  MoveL 1332 to (515.77, 1197.49, 513.19) mm, rotated rx -180 ry 0 rz -88.32 deg; joints [33.086, -49.843, -64.366, 36.804, -42.297, -55.101]
  MoveL 1333 to (513.37, 1199.03, 513.19) mm, rotated rx -180 ry 0 rz -88.32 deg; joints [32.917, -49.844, -64.366, 36.702, -42.2, -54.906]
  MoveL 1334 to (510.99, 1200.59, 513.19) mm, rotated rx -180 ry 0 rz -88.32 deg; joints [32.749, -49.843, -64.366, 36.6, -42.102, -54.711]
  MoveL 1335 to (508.6, 1202.15, 513.19) mm, rotated rx 180 ry 0 rz -88.32 deg; joints [32.58, -49.841, -64.365, 36.498, -42.004, -54.517]
  MoveL 1336 to (506.22, 1203.72, 513.19) mm, rotated rx -180 ry 0 rz -88.32 deg; joints [32.411, -49.837, -64.363, 36.396, -41.905, -54.322]
  MoveL 1337 to (503.85, 1205.29, 513.19) mm, rotated rx 180 ry 0 rz -88.32 deg; joints [32.243, -49.831, -64.361, 36.293, -41.806, -54.128]
  MoveL 1338 to (501.47, 1206.87, 513.19) mm, rotated rx -180 ry 0 rz -88.32 deg; joints [32.074, -49.825, -64.357, 36.19, -41.707, -53.934]
  MoveL 1339 to (499.11, 1208.46, 513.19) mm, rotated rx -180 ry 0 rz -88.32 deg; joints [31.906, -49.816, -64.354, 36.088, -41.607, -53.739]
  MoveL 1340 to (496.75, 1210.05, 513.19) mm, rotated rx -180 ry 0 rz -88.32 deg; joints [31.737, -49.807, -64.349, 35.985, -41.507, -53.545]
  MoveL 1341 to (494.39, 1211.65, 513.19) mm, rotated rx -180 ry 0 rz -88.32 deg; joints [31.569, -49.796, -64.344, 35.881, -41.406, -53.351]
  MoveL 1342 to (492.03, 1213.26, 513.19) mm, rotated rx -180 ry 0 rz -88.32 deg; joints [31.401, -49.783, -64.338, 35.778, -41.305, -53.157]
  MoveL 1343 to (489.69, 1214.88, 513.19) mm, rotated rx -180 ry 0 rz -88.32 deg; joints [31.233, -49.769, -64.332, 35.675, -41.204, -52.963]
  MoveL 1344 to (487.34, 1216.5, 513.19) mm, rotated rx -180 ry 0 rz -88.32 deg; joints [31.064, -49.754, -64.324, 35.571, -41.103, -52.77]
  MoveL 1345 to (485, 1218.12, 513.19) mm, rotated rx -180 ry 0 rz -88.32 deg; joints [30.896, -49.737, -64.316, 35.468, -41.001, -52.576]
  MoveL 1346 to (482.67, 1219.76, 513.19) mm, rotated rx -180 ry 0 rz -88.32 deg; joints [30.728, -49.718, -64.308, 35.364, -40.899, -52.383]
  MoveL 1347 to (480.34, 1221.4, 513.19) mm, rotated rx 180 ry 0 rz -88.32 deg; joints [30.561, -49.698, -64.299, 35.26, -40.796, -52.189]
  MoveL 1348 to (478.01, 1223.04, 513.19) mm, rotated rx -180 ry 0 rz -88.32 deg; joints [30.393, -49.677, -64.289, 35.156, -40.693, -51.996]
  MoveL 1349 to (475.69, 1224.7, 513.19) mm, rotated rx -180 ry 0 rz -88.32 deg; joints [30.225, -49.655, -64.278, 35.052, -40.59, -51.803]
  MoveL 1350 to (473.37, 1226.36, 513.19) mm, rotated rx -180 ry 0 rz -88.32 deg; joints [30.058, -49.631, -64.267, 34.947, -40.487, -51.61]
  MoveL 1351 to (471.06, 1228.02, 513.19) mm, rotated rx 180 ry 0 rz -88.32 deg; joints [29.891, -49.605, -64.255, 34.843, -40.383, -51.418]
  MoveL 1352 to (468.75, 1229.7, 513.19) mm, rotated rx -180 ry 0 rz -88.32 deg; joints [29.723, -49.578, -64.243, 34.739, -40.279, -51.225]
  MoveL 1353 to (466.45, 1231.38, 513.19) mm, rotated rx -180 ry 0 rz -88.32 deg; joints [29.556, -49.55, -64.229, 34.634, -40.175, -51.033]
  MoveL 1354 to (464.15, 1233.06, 513.19) mm, rotated rx -180 ry 0 rz -88.32 deg; joints [29.39, -49.52, -64.216, 34.529, -40.07, -50.841]
  MoveL 1355 to (461.86, 1234.75, 513.19) mm, rotated rx -180 ry 0 rz -88.32 deg; joints [29.223, -49.489, -64.201, 34.425, -39.965, -50.649]
  MoveL 1356 to (459.57, 1236.45, 513.19) mm, rotated rx -180 ry 0 rz -88.32 deg; joints [29.056, -49.456, -64.186, 34.32, -39.86, -50.457]
  MoveL 1357 to (457.29, 1238.16, 513.19) mm, rotated rx -180 ry 0 rz -88.32 deg; joints [28.89, -49.422, -64.17, 34.215, -39.754, -50.265]
  MoveL 1358 to (455.01, 1239.87, 513.19) mm, rotated rx -180 ry 0 rz -88.32 deg; joints [28.724, -49.387, -64.153, 34.11, -39.648, -50.074]
  MoveL 1359 to (452.74, 1241.59, 513.19) mm, rotated rx -180 ry 0 rz -88.32 deg; joints [28.558, -49.35, -64.136, 34.005, -39.542, -49.882]
  MoveL 1360 to (450.47, 1243.31, 513.19) mm, rotated rx -180 ry 0 rz -88.32 deg; joints [28.393, -49.312, -64.118, 33.9, -39.436, -49.691]
  MoveL 1361 to (448.2, 1245.04, 513.19) mm, rotated rx 180 ry 0 rz -88.32 deg; joints [28.227, -49.272, -64.1, 33.794, -39.329, -49.5]
  MoveL 1362 to (445.94, 1246.78, 513.19) mm, rotated rx -180 ry 0 rz -88.32 deg; joints [28.062, -49.231, -64.08, 33.689, -39.223, -49.31]
  MoveL 1363 to (443.69, 1248.52, 513.19) mm, rotated rx -180 ry 0 rz -88.32 deg; joints [27.897, -49.189, -64.061, 33.584, -39.115, -49.119]
  MoveL 1364 to (441.44, 1250.27, 513.19) mm, rotated rx -180 ry 0 rz -88.32 deg; joints [27.732, -49.145, -64.04, 33.478, -39.008, -48.929]
  MoveL 1365 to (439.19, 1252.03, 513.19) mm, rotated rx -180 ry 0 rz -88.32 deg; joints [27.568, -49.1, -64.019, 33.373, -38.901, -48.739]
  MoveL 1366 to (436.95, 1253.79, 513.19) mm, rotated rx 180 ry 0 rz -88.32 deg; joints [27.404, -49.053, -63.997, 33.267, -38.793, -48.549]
  MoveL 1367 to (434.72, 1255.56, 513.19) mm, rotated rx -180 ry 0 rz -88.32 deg; joints [27.24, -49.005, -63.974, 33.162, -38.685, -48.36]
  MoveL 1368 to (432.49, 1257.33, 513.19) mm, rotated rx -180 ry 0 rz -88.32 deg; joints [27.076, -48.956, -63.951, 33.056, -38.577, -48.17]
  MoveL 1369 to (430.26, 1259.11, 513.19) mm, rotated rx -180 ry 0 rz -88.32 deg; joints [26.913, -48.906, -63.927, 32.951, -38.468, -47.981]
  MoveL 1370 to (428.04, 1260.9, 513.19) mm, rotated rx 180 ry 0 rz -88.32 deg; joints [26.749, -48.854, -63.903, 32.845, -38.36, -47.793]
  MoveL 1371 to (425.83, 1262.69, 513.19) mm, rotated rx -180 ry 0 rz -88.32 deg; joints [26.587, -48.8, -63.878, 32.739, -38.251, -47.604]
  MoveL 1372 to (423.62, 1264.49, 513.19) mm, rotated rx -180 ry 0 rz -88.32 deg; joints [26.424, -48.746, -63.852, 32.634, -38.142, -47.416]
  MoveL 1373 to (421.41, 1266.3, 513.19) mm, rotated rx 180 ry 0 rz -88.32 deg; joints [26.262, -48.69, -63.826, 32.528, -38.033, -47.227]
  MoveL 1374 to (419.21, 1268.11, 513.19) mm, rotated rx -180 ry 0 rz -88.32 deg; joints [26.1, -48.633, -63.799, 32.422, -37.924, -47.04]
  MoveL 1375 to (417.02, 1269.93, 513.19) mm, rotated rx -180 ry 0 rz -88.32 deg; joints [25.939, -48.574, -63.771, 32.316, -37.814, -46.852]
  MoveL 1376 to (414.83, 1271.75, 513.19) mm, rotated rx -180 ry 0 rz -88.32 deg; joints [25.777, -48.514, -63.742, 32.21, -37.704, -46.665]
  MoveL 1377 to (412.65, 1273.58, 513.19) mm, rotated rx 180 ry 0 rz -88.32 deg; joints [25.617, -48.453, -63.713, 32.105, -37.594, -46.478]
  MoveL 1378 to (410.47, 1275.42, 513.19) mm, rotated rx -180 ry 0 rz -88.32 deg; joints [25.456, -48.39, -63.684, 31.999, -37.485, -46.291]
  MoveL 1379 to (408.29, 1277.26, 513.19) mm, rotated rx -180 ry 0 rz -88.32 deg; joints [25.296, -48.327, -63.653, 31.893, -37.374, -46.104]
  MoveL 1380 to (406.12, 1279.11, 513.19) mm, rotated rx -180 ry 0 rz -88.32 deg; joints [25.136, -48.262, -63.622, 31.787, -37.264, -45.918]
  MoveL 1381 to (403.96, 1280.97, 513.19) mm, rotated rx -180 ry 0 rz -88.32 deg; joints [24.977, -48.195, -63.591, 31.681, -37.154, -45.732]
  MoveL 1382 to (401.8, 1282.83, 513.19) mm, rotated rx 180 ry 0 rz -88.32 deg; joints [24.818, -48.128, -63.559, 31.575, -37.043, -45.546]
  MoveL 1383 to (399.65, 1284.69, 513.19) mm, rotated rx 180 ry 0 rz -88.32 deg; joints [24.659, -48.059, -63.526, 31.47, -36.933, -45.361]
  MoveL 1384 to (397.5, 1286.57, 513.19) mm, rotated rx -180 ry 0 rz -88.32 deg; joints [24.501, -47.989, -63.492, 31.364, -36.822, -45.176]
  MoveL 1385 to (395.36, 1288.44, 513.19) mm, rotated rx 180 ry 0 rz -88.32 deg; joints [24.343, -47.917, -63.458, 31.258, -36.711, -44.991]
  MoveL 1386 to (393.22, 1290.33, 513.19) mm, rotated rx 180 ry 0 rz -88.32 deg; joints [24.185, -47.845, -63.423, 31.152, -36.6, -44.807]
  MoveL 1387 to (391.09, 1292.22, 513.19) mm, rotated rx -180 ry 0 rz -88.32 deg; joints [24.028, -47.771, -63.388, 31.046, -36.489, -44.622]
  MoveL 1388 to (388.96, 1294.12, 513.19) mm, rotated rx 180 ry 0 rz -88.32 deg; joints [23.872, -47.696, -63.352, 30.941, -36.378, -44.438]
  MoveL 1389 to (386.84, 1296.02, 513.19) mm, rotated rx 180 ry 0 rz -88.32 deg; joints [23.715, -47.619, -63.315, 30.835, -36.267, -44.255]
  MoveL 1390 to (384.72, 1297.93, 513.19) mm, rotated rx 180 ry 0 rz -88.32 deg; joints [23.56, -47.542, -63.278, 30.729, -36.155, -44.072]
  MoveL 1391 to (382.61, 1299.84, 513.19) mm, rotated rx -180 ry 0 rz -88.32 deg; joints [23.404, -47.463, -63.24, 30.624, -36.044, -43.889]
  MoveL 1392 to (380.51, 1301.76, 513.19) mm, rotated rx -180 ry 0 rz -88.32 deg; joints [23.249, -47.383, -63.201, 30.518, -35.932, -43.706]
  MoveL 1393 to (378.41, 1303.69, 513.19) mm, rotated rx 180 ry 0 rz -88.32 deg; joints [23.095, -47.302, -63.162, 30.412, -35.821, -43.524]
  MoveL 1394 to (376.31, 1305.62, 513.19) mm, rotated rx -180 ry 0 rz -88.32 deg; joints [22.941, -47.22, -63.123, 30.307, -35.709, -43.341]
  MoveL 1395 to (374.22, 1307.56, 513.19) mm, rotated rx -180 ry 0 rz -88.32 deg; joints [22.787, -47.137, -63.082, 30.201, -35.598, -43.16]
  MoveL 1396 to (372.14, 1309.51, 513.19) mm, rotated rx -180 ry 0 rz -88.32 deg; joints [22.634, -47.052, -63.041, 30.096, -35.486, -42.978]
  MoveL 1397 to (370.06, 1311.46, 513.19) mm, rotated rx 180 ry 0 rz -88.32 deg; joints [22.481, -46.966, -62.999, 29.991, -35.375, -42.797]
  MoveL 1398 to (367.99, 1313.41, 513.19) mm, rotated rx 180 ry 0 rz -88.32 deg; joints [22.329, -46.879, -62.957, 29.885, -35.263, -42.617]
  MoveL 1399 to (365.92, 1315.37, 513.19) mm, rotated rx -180 ry 0 rz -88.32 deg; joints [22.177, -46.791, -62.914, 29.78, -35.151, -42.436]
  MoveL 1400 to (363.86, 1317.34, 513.19) mm, rotated rx -180 ry 0 rz -88.32 deg; joints [22.026, -46.702, -62.871, 29.675, -35.039, -42.256]
  MoveL 1401 to (361.8, 1319.31, 513.19) mm, rotated rx 180 ry 0 rz -88.32 deg; joints [21.875, -46.612, -62.827, 29.569, -34.928, -42.076]
  MoveL 1402 to (359.75, 1321.29, 513.19) mm, rotated rx -180 ry 0 rz -88.32 deg; joints [21.725, -46.521, -62.782, 29.464, -34.816, -41.897]
  MoveL 1403 to (357.71, 1323.28, 513.19) mm, rotated rx 180 ry 0 rz -88.32 deg; joints [21.575, -46.428, -62.737, 29.359, -34.704, -41.718]
  MoveL 1404 to (355.67, 1325.27, 513.19) mm, rotated rx 180 ry 0 rz -88.32 deg; joints [21.426, -46.335, -62.691, 29.254, -34.593, -41.539]
  MoveL 1405 to (353.63, 1327.26, 513.19) mm, rotated rx 180 ry 0 rz -88.32 deg; joints [21.277, -46.24, -62.644, 29.149, -34.481, -41.361]
  MoveL 1406 to (351.6, 1329.27, 513.19) mm, rotated rx -180 ry 0 rz -88.32 deg; joints [21.129, -46.144, -62.597, 29.044, -34.369, -41.183]
  MoveL 1407 to (349.58, 1331.27, 513.19) mm, rotated rx 180 ry 0 rz -88.32 deg; joints [20.981, -46.047, -62.55, 28.94, -34.258, -41.005]
  MoveL 1408 to (347.56, 1333.29, 513.19) mm, rotated rx 180 ry 0 rz -88.32 deg; joints [20.834, -45.95, -62.501, 28.835, -34.146, -40.828]
  MoveL 1409 to (345.55, 1335.3, 513.19) mm, rotated rx -180 ry 0 rz -88.32 deg; joints [20.687, -45.851, -62.453, 28.73, -34.035, -40.651]
  MoveL 1410 to (343.55, 1337.33, 513.19) mm, rotated rx -180 ry 0 rz -88.32 deg; joints [20.541, -45.751, -62.403, 28.626, -33.923, -40.475]
  MoveL 1411 to (341.55, 1339.36, 513.19) mm, rotated rx -180 ry 0 rz -88.32 deg; joints [20.395, -45.65, -62.353, 28.521, -33.812, -40.298]
  MoveL 1412 to (339.55, 1341.39, 513.19) mm, rotated rx -180 ry 0 rz -88.32 deg; joints [20.25, -45.548, -62.302, 28.417, -33.7, -40.123]
  MoveL 1413 to (337.56, 1343.44, 513.19) mm, rotated rx -180 ry 0 rz -88.32 deg; joints [20.106, -45.445, -62.251, 28.312, -33.589, -39.947]
  MoveL 1414 to (335.58, 1345.48, 513.19) mm, rotated rx -180 ry 0 rz -88.32 deg; joints [19.962, -45.341, -62.199, 28.208, -33.478, -39.772]
  MoveL 1415 to (333.6, 1347.54, 513.19) mm, rotated rx -180 ry 0 rz -88.32 deg; joints [19.818, -45.236, -62.147, 28.104, -33.367, -39.597]
  MoveL 1416 to (331.63, 1349.59, 513.19) mm, rotated rx -180 ry 0 rz -88.32 deg; joints [19.675, -45.13, -62.094, 28, -33.256, -39.423]
  MoveL 1417 to (329.67, 1351.66, 513.19) mm, rotated rx 180 ry 0 rz -88.32 deg; joints [19.533, -45.023, -62.041, 27.896, -33.145, -39.249]
  MoveL 1418 to (327.71, 1353.73, 513.19) mm, rotated rx 180 ry 0 rz -88.32 deg; joints [19.391, -44.915, -61.986, 27.792, -33.034, -39.075]
  MoveL 1419 to (325.75, 1355.8, 513.19) mm, rotated rx -180 ry 0 rz -88.32 deg; joints [19.25, -44.806, -61.932, 27.688, -32.923, -38.902]
  MoveL 1420 to (323.8, 1357.88, 513.19) mm, rotated rx -180 ry 0 rz -88.32 deg; joints [19.109, -44.697, -61.876, 27.585, -32.812, -38.729]
  MoveL 1421 to (321.86, 1359.96, 513.19) mm, rotated rx -180 ry 0 rz -88.32 deg; joints [18.969, -44.586, -61.821, 27.481, -32.702, -38.557]
  MoveL 1422 to (319.92, 1362.06, 513.19) mm, rotated rx 180 ry 0 rz -88.32 deg; joints [18.829, -44.474, -61.764, 27.377, -32.591, -38.385]
  MoveL 1423 to (317.99, 1364.15, 513.19) mm, rotated rx -180 ry 0 rz -88.32 deg; joints [18.69, -44.362, -61.707, 27.274, -32.481, -38.213]
  MoveL 1424 to (316.07, 1366.25, 513.19) mm, rotated rx -180 ry 0 rz -88.32 deg; joints [18.552, -44.248, -61.65, 27.171, -32.371, -38.042]
  MoveL 1425 to (314.15, 1368.36, 513.19) mm, rotated rx -180 ry 0 rz -88.32 deg; joints [18.414, -44.134, -61.592, 27.068, -32.261, -37.871]
  MoveL 1426 to (312.24, 1370.47, 513.19) mm, rotated rx 180 ry 0 rz -88.32 deg; joints [18.277, -44.019, -61.533, 26.965, -32.151, -37.7]
  MoveL 1427 to (310.33, 1372.59, 513.19) mm, rotated rx 180 ry 0 rz -88.32 deg; joints [18.141, -43.903, -61.474, 26.862, -32.041, -37.53]
  MoveL 1428 to (308.43, 1374.71, 513.19) mm, rotated rx -180 ry 0 rz -88.32 deg; joints [18.005, -43.786, -61.414, 26.759, -31.932, -37.361]
  MoveL 1429 to (306.53, 1376.84, 513.19) mm, rotated rx 180 ry 0 rz -88.32 deg; joints [17.869, -43.668, -61.354, 26.656, -31.822, -37.191]
  MoveL 1430 to (304.64, 1378.98, 513.19) mm, rotated rx 180 ry 0 rz -88.32 deg; joints [17.734, -43.549, -61.293, 26.554, -31.713, -37.022]
  MoveL 1431 to (302.76, 1381.11, 513.19) mm, rotated rx 180 ry 0 rz -88.32 deg; joints [17.6, -43.43, -61.232, 26.451, -31.604, -36.854]
  MoveL 1432 to (300.88, 1383.26, 513.19) mm, rotated rx -180 ry 0 rz -88.32 deg; joints [17.466, -43.309, -61.17, 26.349, -31.495, -36.686]
  MoveL 1433 to (299.01, 1385.41, 513.19) mm, rotated rx -180 ry 0 rz -88.32 deg; joints [17.333, -43.188, -61.107, 26.247, -31.387, -36.518]
  MoveL 1434 to (297.15, 1387.56, 513.19) mm, rotated rx -180 ry 0 rz -88.32 deg; joints [17.201, -43.066, -61.044, 26.144, -31.278, -36.351]
  MoveL 1435 to (295.29, 1389.72, 513.19) mm, rotated rx -180 ry 0 rz -88.32 deg; joints [17.069, -42.944, -60.981, 26.042, -31.17, -36.184]
  MoveL 1436 to (293.44, 1391.89, 513.19) mm, rotated rx -180 ry 0 rz -88.32 deg; joints [16.938, -42.82, -60.917, 25.941, -31.062, -36.017]
  MoveL 1437 to (291.59, 1394.06, 513.19) mm, rotated rx -180 ry 0 rz -88.32 deg; joints [16.808, -42.696, -60.852, 25.839, -30.954, -35.851]
  MoveL 1438 to (289.75, 1396.23, 513.19) mm, rotated rx 180 ry 0 rz -88.32 deg; joints [16.678, -42.571, -60.787, 25.737, -30.846, -35.686]
  MoveL 1439 to (287.91, 1398.41, 513.19) mm, rotated rx 180 ry 0 rz -88.32 deg; joints [16.548, -42.445, -60.721, 25.636, -30.739, -35.521]
  MoveL 1440 to (286.08, 1400.6, 513.19) mm, rotated rx 180 ry 0 rz -88.32 deg; joints [16.42, -42.318, -60.655, 25.535, -30.631, -35.356]
  MoveL 1441 to (284.26, 1402.79, 513.19) mm, rotated rx 180 ry 0 rz -88.32 deg; joints [16.292, -42.191, -60.588, 25.433, -30.524, -35.191]
  MoveL 1442 to (282.45, 1404.99, 513.19) mm, rotated rx -180 ry 0 rz -88.32 deg; joints [16.164, -42.063, -60.521, 25.332, -30.418, -35.027]
  MoveL 1443 to (280.64, 1407.19, 513.19) mm, rotated rx -180 ry 0 rz -88.32 deg; joints [16.037, -41.934, -60.453, 25.231, -30.311, -34.864]
  MoveL 1444 to (278.83, 1409.4, 513.19) mm, rotated rx -180 ry 0 rz -88.32 deg; joints [15.911, -41.804, -60.385, 25.131, -30.205, -34.701]
  MoveL 1445 to (277.03, 1411.61, 513.19) mm, rotated rx -180 ry 0 rz -88.32 deg; joints [15.786, -41.674, -60.316, 25.03, -30.099, -34.538]
  MoveL 1446 to (275.24, 1413.82, 513.19) mm, rotated rx -180 ry 0 rz -88.32 deg; joints [15.661, -41.543, -60.247, 24.93, -29.993, -34.376]
  MoveL 1447 to (273.46, 1416.04, 513.19) mm, rotated rx 180 ry 0 rz -88.32 deg; joints [15.536, -41.412, -60.177, 24.829, -29.887, -34.214]
  MoveL 1448 to (271.68, 1418.27, 513.19) mm, rotated rx -180 ry 0 rz -88.32 deg; joints [15.413, -41.279, -60.107, 24.729, -29.782, -34.052]
  MoveL 1449 to (269.91, 1420.5, 513.19) mm, rotated rx -180 ry 0 rz -88.32 deg; joints [15.29, -41.147, -60.036, 24.629, -29.677, -33.891]
  MoveL 1450 to (268.14, 1422.74, 513.19) mm, rotated rx 180 ry 0 rz -88.32 deg; joints [15.167, -41.013, -59.965, 24.529, -29.572, -33.731]
  MoveL 1451 to (266.38, 1424.98, 513.19) mm, rotated rx -180 ry 0 rz -88.32 deg; joints [15.046, -40.879, -59.893, 24.429, -29.468, -33.571]
  MoveL 1452 to (264.62, 1427.23, 513.19) mm, rotated rx -180 ry 0 rz -88.32 deg; joints [14.925, -40.744, -59.821, 24.33, -29.363, -33.411]
  MoveL 1453 to (262.88, 1429.48, 513.19) mm, rotated rx 180 ry 0 rz -88.32 deg; joints [14.804, -40.608, -59.748, 24.23, -29.26, -33.252]
  MoveL 1454 to (261.14, 1431.73, 513.19) mm, rotated rx 180 ry 0 rz -88.32 deg; joints [14.684, -40.472, -59.674, 24.131, -29.156, -33.093]
  MoveL 1455 to (259.4, 1433.99, 513.19) mm, rotated rx -180 ry 0 rz -88.32 deg; joints [14.565, -40.335, -59.601, 24.032, -29.053, -32.935]
  MoveL 1456 to (257.67, 1436.26, 513.19) mm, rotated rx 180 ry 0 rz -88.32 deg; joints [14.447, -40.198, -59.526, 23.933, -28.949, -32.777]
  MoveL 1457 to (255.95, 1438.53, 513.19) mm, rotated rx -180 ry 0 rz -88.32 deg; joints [14.329, -40.06, -59.452, 23.834, -28.847, -32.619]
  MoveL 1458 to (254.23, 1440.8, 513.19) mm, rotated rx 180 ry 0 rz -88.32 deg; joints [14.212, -39.922, -59.376, 23.736, -28.744, -32.462]
  MoveL 1459 to (252.52, 1443.08, 513.19) mm, rotated rx -180 ry 0 rz -88.32 deg; joints [14.095, -39.783, -59.301, 23.637, -28.642, -32.306]
  MoveL 1460 to (250.82, 1445.37, 513.19) mm, rotated rx 180 ry 0 rz -88.32 deg; joints [13.979, -39.643, -59.224, 23.539, -28.54, -32.149]
  MoveL 1461 to (249.12, 1447.66, 513.19) mm, rotated rx 180 ry 0 rz -88.32 deg; joints [13.864, -39.503, -59.148, 23.441, -28.439, -31.994]
  MoveL 1462 to (247.43, 1449.95, 513.19) mm, rotated rx -180 ry 0 rz -88.32 deg; joints [13.749, -39.362, -59.07, 23.343, -28.338, -31.838]
  MoveL 1463 to (245.75, 1452.25, 513.19) mm, rotated rx -180 ry 0 rz -88.32 deg; joints [13.635, -39.221, -58.993, 23.245, -28.237, -31.684]
  MoveL 1464 to (244.07, 1454.56, 513.19) mm, rotated rx 180 ry 0 rz -88.32 deg; joints [13.522, -39.079, -58.915, 23.147, -28.136, -31.529]
  MoveL 1465 to (242.4, 1456.87, 513.19) mm, rotated rx 180 ry 0 rz -88.32 deg; joints [13.409, -38.937, -58.836, 23.05, -28.036, -31.375]
  MoveL 1466 to (240.74, 1459.18, 513.19) mm, rotated rx 180 ry 0 rz -88.32 deg; joints [13.297, -38.794, -58.757, 22.952, -27.936, -31.222]
  MoveL 1467 to (239.08, 1461.5, 513.19) mm, rotated rx 180 ry 0 rz -88.32 deg; joints [13.186, -38.65, -58.678, 22.855, -27.836, -31.069]
  MoveL 1468 to (237.43, 1463.82, 513.19) mm, rotated rx -180 ry 0 rz -88.32 deg; joints [13.075, -38.507, -58.598, 22.758, -27.737, -30.917]
  MoveL 1469 to (235.78, 1466.15, 513.19) mm, rotated rx 180 ry 0 rz -88.32 deg; joints [12.965, -38.362, -58.517, 22.661, -27.638, -30.764]
  MoveL 1470 to (234.14, 1468.48, 513.19) mm, rotated rx 180 ry 0 rz -88.32 deg; joints [12.856, -38.217, -58.436, 22.565, -27.54, -30.613]
  MoveL 1471 to (232.51, 1470.81, 513.19) mm, rotated rx 180 ry 0 rz -88.32 deg; joints [12.747, -38.072, -58.355, 22.468, -27.442, -30.462]
  MoveL 1472 to (230.89, 1473.16, 513.19) mm, rotated rx 180 ry 0 rz -88.32 deg; joints [12.639, -37.926, -58.273, 22.372, -27.344, -30.311]
  MoveL 1473 to (229.27, 1475.5, 513.19) mm, rotated rx 180 ry 0 rz -88.32 deg; joints [12.531, -37.78, -58.191, 22.276, -27.247, -30.161]
  MoveL 1474 to (227.66, 1477.85, 513.19) mm, rotated rx 180 ry 0 rz -88.32 deg; joints [12.425, -37.633, -58.108, 22.18, -27.149, -30.011]
  MoveL 1475 to (226.05, 1480.21, 513.19) mm, rotated rx -180 ry 0 rz -88.32 deg; joints [12.319, -37.486, -58.025, 22.085, -27.053, -29.862]
  MoveL 1476 to (224.45, 1482.57, 513.19) mm, rotated rx -180 ry 0 rz -88.32 deg; joints [12.213, -37.339, -57.942, 21.989, -26.956, -29.713]
  MoveL 1477 to (222.86, 1484.93, 513.19) mm, rotated rx -180 ry 0 rz -88.32 deg; joints [12.108, -37.191, -57.858, 21.894, -26.86, -29.565]
  MoveL 1478 to (221.27, 1487.3, 513.19) mm, rotated rx 180 ry 0 rz -88.32 deg; joints [12.004, -37.043, -57.773, 21.799, -26.765, -29.417]
  MoveL 1479 to (219.69, 1489.67, 513.19) mm, rotated rx 180 ry 0 rz -88.32 deg; joints [11.901, -36.894, -57.688, 21.704, -26.67, -29.27]
  MoveL 1480 to (218.12, 1492.05, 513.19) mm, rotated rx -180 ry 0 rz -88.32 deg; joints [11.798, -36.745, -57.603, 21.609, -26.575, -29.123]
  MoveL 1481 to (216.56, 1494.43, 513.19) mm, rotated rx -180 ry 0 rz -88.32 deg; joints [11.695, -36.595, -57.517, 21.515, -26.48, -28.977]
  MoveL 1482 to (215, 1496.81, 513.19) mm, rotated rx -180 ry 0 rz -88.32 deg; joints [11.594, -36.445, -57.431, 21.42, -26.386, -28.831]
  MoveL 1483 to (213.45, 1499.2, 513.19) mm, rotated rx 180 ry 0 rz -88.32 deg; joints [11.493, -36.295, -57.344, 21.326, -26.293, -28.685]
  MoveL 1484 to (211.9, 1501.6, 513.19) mm, rotated rx -180 ry 0 rz -88.32 deg; joints [11.393, -36.144, -57.257, 21.232, -26.199, -28.54]
  MoveL 1485 to (210.36, 1504, 513.19) mm, rotated rx -180 ry 0 rz -88.32 deg; joints [11.293, -35.993, -57.17, 21.139, -26.106, -28.396]
  MoveL 1486 to (208.83, 1506.4, 513.19) mm, rotated rx 180 ry 0 rz -88.32 deg; joints [11.194, -35.842, -57.082, 21.045, -26.014, -28.252]
  MoveL 1487 to (207.3, 1508.81, 513.19) mm, rotated rx 180 ry 0 rz -88.32 deg; joints [11.096, -35.69, -56.994, 20.952, -25.922, -28.108]
  MoveL 1488 to (205.78, 1511.22, 513.19) mm, rotated rx -180 ry 0 rz -88.32 deg; joints [10.998, -35.538, -56.905, 20.859, -25.83, -27.965]
  MoveL 1489 to (204.27, 1513.63, 513.19) mm, rotated rx 180 ry 0 rz -88.32 deg; joints [10.901, -35.386, -56.816, 20.766, -25.739, -27.823]
  MoveL 1490 to (202.77, 1516.05, 513.19) mm, rotated rx -180 ry 0 rz -88.32 deg; joints [10.804, -35.233, -56.727, 20.673, -25.648, -27.681]
  MoveL 1491 to (201.27, 1518.48, 513.19) mm, rotated rx -180 ry 0 rz -88.32 deg; joints [10.709, -35.08, -56.637, 20.581, -25.558, -27.54]
  MoveL 1492 to (199.78, 1520.91, 513.19) mm, rotated rx -180 ry 0 rz -88.32 deg; joints [10.614, -34.926, -56.546, 20.488, -25.468, -27.399]
  MoveL 1493 to (198.29, 1523.34, 513.19) mm, rotated rx 180 ry 0 rz -88.32 deg; joints [10.519, -34.773, -56.456, 20.396, -25.378, -27.258]
  MoveL 1494 to (196.82, 1525.78, 513.19) mm, rotated rx -180 ry 0 rz -88.32 deg; joints [10.425, -34.619, -56.364, 20.305, -25.289, -27.118]
  MoveL 1495 to (195.34, 1528.22, 513.19) mm, rotated rx 180 ry 0 rz -88.32 deg; joints [10.332, -34.465, -56.273, 20.213, -25.2, -26.979]
  MoveL 1496 to (193.88, 1530.66, 513.19) mm, rotated rx 180 ry 0 rz -88.32 deg; joints [10.24, -34.31, -56.181, 20.122, -25.111, -26.84]
  MoveL 1497 to (192.42, 1533.11, 513.19) mm, rotated rx 180 ry 0 rz -88.32 deg; joints [10.148, -34.155, -56.089, 20.031, -25.024, -26.701]
  MoveL 1498 to (190.97, 1535.56, 513.19) mm, rotated rx -180 ry 0 rz -88.32 deg; joints [10.056, -34, -55.996, 19.94, -24.936, -26.563]
  MoveL 1499 to (189.53, 1538.02, 513.19) mm, rotated rx -180 ry 0 rz -88.32 deg; joints [9.966, -33.845, -55.903, 19.849, -24.849, -26.426]
  MoveL 1500 to (188.09, 1540.48, 513.19) mm, rotated rx 180 ry 0 rz -88.32 deg; joints [9.876, -33.689, -55.809, 19.759, -24.762, -26.289]
  MoveL 1501 to (186.66, 1542.95, 513.19) mm, rotated rx -180 ry 0 rz -88.32 deg; joints [9.786, -33.533, -55.716, 19.668, -24.676, -26.153]
  MoveL 1502 to (185.24, 1545.42, 513.19) mm, rotated rx -180 ry 0 rz -88.32 deg; joints [9.697, -33.377, -55.621, 19.579, -24.59, -26.017]
  MoveL 1503 to (183.82, 1547.89, 513.19) mm, rotated rx 180 ry 0 rz -88.32 deg; joints [9.609, -33.221, -55.527, 19.489, -24.505, -25.881]
  MoveL 1504 to (182.41, 1550.37, 513.19) mm, rotated rx 180 ry 0 rz -88.32 deg; joints [9.522, -33.065, -55.432, 19.399, -24.42, -25.747]
  MoveL 1505 to (181.01, 1552.85, 513.19) mm, rotated rx 180 ry 0 rz -88.32 deg; joints [9.435, -32.908, -55.336, 19.31, -24.335, -25.612]
  MoveL 1506 to (179.62, 1555.33, 513.19) mm, rotated rx 180 ry 0 rz -88.32 deg; joints [9.349, -32.751, -55.241, 19.221, -24.251, -25.478]
  MoveL 1507 to (178.23, 1557.82, 513.19) mm, rotated rx 180 ry 0 rz -88.32 deg; joints [9.263, -32.594, -55.144, 19.132, -24.168, -25.345]
  MoveL 1508 to (176.85, 1560.31, 513.19) mm, rotated rx 180 ry 0 rz -88.32 deg; joints [9.178, -32.436, -55.048, 19.044, -24.084, -25.212]
  MoveL 1509 to (175.47, 1562.81, 513.19) mm, rotated rx 180 ry 0 rz -88.32 deg; joints [9.094, -32.279, -54.951, 18.956, -24.002, -25.08]
  MoveL 1510 to (174.11, 1565.31, 513.19) mm, rotated rx 180 ry 0 rz -88.32 deg; joints [9.01, -32.121, -54.854, 18.868, -23.919, -24.949]
  MoveL 1511 to (172.75, 1567.82, 513.19) mm, rotated rx -180 ry 0 rz -88.32 deg; joints [8.927, -31.963, -54.756, 18.78, -23.837, -24.818]
  MoveL 1512 to (171.39, 1570.32, 513.19) mm, rotated rx -180 ry 0 rz -88.32 deg; joints [8.844, -31.805, -54.658, 18.692, -23.756, -24.687]
  MoveL 1513 to (170.05, 1572.84, 513.19) mm, rotated rx -180 ry 0 rz -88.32 deg; joints [8.763, -31.646, -54.56, 18.605, -23.675, -24.557]
  MoveL 1514 to (168.71, 1575.35, 513.19) mm, rotated rx 180 ry 0 rz -88.32 deg; joints [8.681, -31.488, -54.461, 18.518, -23.594, -24.427]
  MoveL 1515 to (167.38, 1577.87, 513.19) mm, rotated rx 180 ry 0 rz -88.32 deg; joints [8.601, -31.329, -54.362, 18.432, -23.514, -24.299]
  MoveL 1516 to (166.05, 1580.4, 513.19) mm, rotated rx -180 ry 0 rz -88.32 deg; joints [8.521, -31.17, -54.263, 18.345, -23.435, -24.17]
  MoveL 1517 to (164.74, 1582.92, 513.19) mm, rotated rx -180 ry 0 rz -88.32 deg; joints [8.441, -31.011, -54.163, 18.259, -23.356, -24.042]
  MoveL 1518 to (163.43, 1585.45, 513.19) mm, rotated rx -180 ry 0 rz -88.32 deg; joints [8.362, -30.852, -54.063, 18.173, -23.277, -23.915]
  MoveL 1519 to (162.12, 1587.99, 513.19) mm, rotated rx 180 ry 0 rz -88.32 deg; joints [8.284, -30.693, -53.963, 18.088, -23.199, -23.788]
  MoveL 1520 to (160.83, 1590.53, 513.19) mm, rotated rx 180 ry 0 rz -88.32 deg; joints [8.206, -30.534, -53.862, 18.002, -23.121, -23.662]
  MoveL 1521 to (159.54, 1593.07, 513.19) mm, rotated rx 180 ry 0 rz -88.32 deg; joints [8.129, -30.374, -53.761, 17.917, -23.043, -23.536]
  MoveL 1522 to (158.25, 1595.61, 513.19) mm, rotated rx 180 ry 0 rz -88.32 deg; joints [8.053, -30.215, -53.659, 17.833, -22.967, -23.411]
  MoveL 1523 to (156.98, 1598.16, 513.19) mm, rotated rx -180 ry 0 rz -88.32 deg; joints [7.977, -30.055, -53.557, 17.748, -22.89, -23.287]
  MoveL 1524 to (155.71, 1600.71, 513.19) mm, rotated rx 180 ry 0 rz -88.32 deg; joints [7.902, -29.895, -53.455, 17.664, -22.814, -23.163]
  MoveL 1525 to (154.45, 1603.27, 513.19) mm, rotated rx 180 ry 0 rz -88.32 deg; joints [7.827, -29.735, -53.353, 17.58, -22.739, -23.04]
  MoveL 1526 to (153.2, 1605.83, 513.19) mm, rotated rx -180 ry 0 rz -88.32 deg; joints [7.753, -29.575, -53.25, 17.496, -22.663, -22.917]
  MoveL 1527 to (151.95, 1608.39, 513.19) mm, rotated rx 180 ry 0 rz -88.32 deg; joints [7.68, -29.415, -53.147, 17.413, -22.589, -22.795]
  MoveL 1528 to (150.71, 1610.96, 513.19) mm, rotated rx -180 ry 0 rz -88.32 deg; joints [7.607, -29.254, -53.043, 17.33, -22.515, -22.673]
  MoveL 1529 to (149.48, 1613.53, 513.19) mm, rotated rx 180 ry 0 rz -88.32 deg; joints [7.535, -29.094, -52.939, 17.247, -22.441, -22.552]
  MoveL 1530 to (148.26, 1616.1, 513.19) mm, rotated rx 180 ry 0 rz -88.32 deg; joints [7.463, -28.933, -52.835, 17.165, -22.368, -22.431]
  MoveL 1531 to (147.04, 1618.68, 513.19) mm, rotated rx 180 ry 0 rz -88.32 deg; joints [7.392, -28.773, -52.731, 17.083, -22.295, -22.311]
  MoveL 1532 to (145.83, 1621.26, 513.19) mm, rotated rx -180 ry 0 rz -88.32 deg; joints [7.322, -28.612, -52.626, 17.001, -22.223, -22.192]
  MoveL 1533 to (144.62, 1623.84, 513.19) mm, rotated rx -180 ry 0 rz -88.32 deg; joints [7.252, -28.451, -52.521, 16.92, -22.151, -22.073]
  MoveL 1534 to (143.43, 1626.43, 513.19) mm, rotated rx 180 ry 0 rz -88.32 deg; joints [7.182, -28.291, -52.416, 16.839, -22.079, -21.955]
  MoveL 1535 to (142.24, 1629.02, 513.19) mm, rotated rx 180 ry 0 rz -88.32 deg; joints [7.114, -28.13, -52.31, 16.758, -22.009, -21.838]
  MoveL 1536 to (141.06, 1631.61, 513.19) mm, rotated rx -180 ry 0 rz -88.32 deg; joints [7.045, -27.969, -52.204, 16.677, -21.938, -21.721]
  MoveL 1537 to (139.89, 1634.21, 513.19) mm, rotated rx 180 ry 0 rz -88.32 deg; joints [6.978, -27.808, -52.098, 16.597, -21.868, -21.604]
  MoveL 1538 to (138.72, 1636.81, 513.19) mm, rotated rx -180 ry 0 rz -88.32 deg; joints [6.911, -27.647, -51.991, 16.517, -21.799, -21.489]
  MoveL 1539 to (137.56, 1639.41, 513.19) mm, rotated rx 180 ry 0 rz -88.32 deg; joints [6.844, -27.486, -51.884, 16.438, -21.73, -21.373]
  MoveL 1540 to (136.41, 1642.02, 513.19) mm, rotated rx -180 ry 0 rz -88.32 deg; joints [6.778, -27.325, -51.777, 16.358, -21.661, -21.259]
  MoveL 1541 to (135.26, 1644.63, 513.19) mm, rotated rx 180 ry 0 rz -88.32 deg; joints [6.713, -27.163, -51.669, 16.28, -21.593, -21.145]
  MoveL 1542 to (134.13, 1647.24, 513.19) mm, rotated rx -180 ry 0 rz -88.32 deg; joints [6.648, -27.002, -51.561, 16.201, -21.525, -21.032]
  MoveL 1543 to (133, 1649.86, 513.19) mm, rotated rx 180 ry 0 rz -88.32 deg; joints [6.584, -26.841, -51.453, 16.123, -21.458, -20.919]
  MoveL 1544 to (131.87, 1652.48, 513.19) mm, rotated rx -180 ry 0 rz -88.32 deg; joints [6.521, -26.68, -51.345, 16.045, -21.391, -20.807]
  MoveL 1545 to (130.76, 1655.1, 513.19) mm, rotated rx 180 ry 0 rz -88.32 deg; joints [6.457, -26.518, -51.236, 15.968, -21.325, -20.695]
  MoveL 1546 to (129.65, 1657.73, 513.19) mm, rotated rx -180 ry 0 rz -88.32 deg; joints [6.395, -26.357, -51.127, 15.89, -21.259, -20.584]
  MoveL 1547 to (128.55, 1660.35, 513.19) mm, rotated rx -180 ry 0 rz -88.32 deg; joints [6.333, -26.196, -51.017, 15.814, -21.194, -20.474]
  MoveL 1548 to (127.46, 1662.99, 513.19) mm, rotated rx 180 ry 0 rz -88.32 deg; joints [6.272, -26.034, -50.908, 15.737, -21.129, -20.364]
  MoveL 1549 to (126.37, 1665.62, 513.19) mm, rotated rx 180 ry 0 rz -88.32 deg; joints [6.211, -25.873, -50.798, 15.661, -21.064, -20.255]
  MoveL 1550 to (125.29, 1668.26, 513.19) mm, rotated rx -180 ry 0 rz -88.32 deg; joints [6.15, -25.712, -50.687, 15.585, -21, -20.147]
  MoveL 1551 to (124.22, 1670.9, 513.19) mm, rotated rx 180 ry 0 rz -88.32 deg; joints [6.091, -25.55, -50.577, 15.51, -20.937, -20.039]
  MoveL 1552 to (123.16, 1673.54, 513.19) mm, rotated rx 180 ry 0 rz -88.32 deg; joints [6.031, -25.389, -50.466, 15.435, -20.874, -19.932]
  MoveL 1553 to (122.1, 1676.19, 513.19) mm, rotated rx 180 ry 0 rz -88.32 deg; joints [5.973, -25.228, -50.355, 15.36, -20.811, -19.826]
  MoveL 1554 to (121.05, 1678.84, 513.19) mm, rotated rx -180 ry 0 rz -88.32 deg; joints [5.915, -25.066, -50.244, 15.286, -20.749, -19.72]
  MoveL 1555 to (120.01, 1681.49, 513.19) mm, rotated rx 180 ry 0 rz -88.32 deg; joints [5.857, -24.905, -50.132, 15.212, -20.688, -19.615]
  MoveL 1556 to (118.98, 1684.15, 513.19) mm, rotated rx -180 ry 0 rz -88.32 deg; joints [5.8, -24.744, -50.02, 15.139, -20.626, -19.51]
  MoveL 1557 to (117.95, 1686.81, 513.19) mm, rotated rx 180 ry 0 rz -88.32 deg; joints [5.743, -24.582, -49.908, 15.066, -20.566, -19.406]
  MoveL 1558 to (116.93, 1689.47, 513.19) mm, rotated rx -180 ry 0 rz -88.32 deg; joints [5.687, -24.421, -49.795, 14.993, -20.505, -19.303]
  MoveL 1559 to (115.92, 1692.13, 513.19) mm, rotated rx -180 ry 0 rz -88.32 deg; joints [5.632, -24.26, -49.683, 14.921, -20.446, -19.2]
  MoveL 1560 to (114.91, 1694.8, 513.19) mm, rotated rx -180 ry 0 rz -88.32 deg; joints [5.577, -24.098, -49.57, 14.849, -20.386, -19.098]
  MoveL 1561 to (113.92, 1697.47, 513.19) mm, rotated rx -180 ry 0 rz -88.32 deg; joints [5.522, -23.937, -49.456, 14.777, -20.327, -18.997]
  MoveL 1562 to (112.93, 1700.14, 513.19) mm, rotated rx -180 ry 0 rz -88.32 deg; joints [5.469, -23.776, -49.343, 14.706, -20.269, -18.896]
  MoveL 1563 to (111.95, 1702.82, 513.19) mm, rotated rx 180 ry 0 rz -88.32 deg; joints [5.415, -23.615, -49.229, 14.635, -20.211, -18.797]
  MoveL 1564 to (110.97, 1705.5, 513.19) mm, rotated rx -180 ry 0 rz -88.32 deg; joints [5.362, -23.454, -49.115, 14.565, -20.153, -18.697]
  MoveL 1565 to (110.01, 1708.18, 513.19) mm, rotated rx 180 ry 0 rz -88.32 deg; joints [5.31, -23.293, -49, 14.495, -20.096, -18.599]
  MoveL 1566 to (109.05, 1710.86, 513.19) mm, rotated rx -180 ry 0 rz -88.32 deg; joints [5.258, -23.132, -48.886, 14.426, -20.04, -18.501]
  MoveL 1567 to (108.1, 1713.55, 513.19) mm, rotated rx 180 ry 0 rz -88.32 deg; joints [5.207, -22.971, -48.771, 14.356, -19.984, -18.403]
  MoveL 1568 to (107.15, 1716.24, 513.19) mm, rotated rx 180 ry 0 rz -88.32 deg; joints [5.156, -22.81, -48.656, 14.288, -19.928, -18.307]
  MoveL 1569 to (106.22, 1718.93, 513.19) mm, rotated rx 180 ry 0 rz -88.32 deg; joints [5.106, -22.649, -48.54, 14.219, -19.873, -18.211]
  MoveL 1570 to (105.29, 1721.62, 513.19) mm, rotated rx 180 ry 0 rz -88.32 deg; joints [5.056, -22.488, -48.425, 14.152, -19.818, -18.116]
  MoveL 1571 to (104.37, 1724.32, 513.19) mm, rotated rx 180 ry 0 rz -88.32 deg; joints [5.007, -22.327, -48.309, 14.084, -19.764, -18.021]
  MoveL 1572 to (103.45, 1727.02, 513.19) mm, rotated rx -180 ry 0 rz -88.32 deg; joints [4.958, -22.166, -48.193, 14.017, -19.71, -17.927]
  MoveL 1573 to (102.55, 1729.72, 513.19) mm, rotated rx -180 ry 0 rz -88.32 deg; joints [4.91, -22.006, -48.076, 13.951, -19.656, -17.834]
  MoveL 1574 to (101.65, 1732.43, 513.19) mm, rotated rx 180 ry 0 rz -88.32 deg; joints [4.862, -21.845, -47.96, 13.885, -19.603, -17.741]
  MoveL 1575 to (100.76, 1735.13, 513.19) mm, rotated rx -180 ry 0 rz -88.32 deg; joints [4.815, -21.685, -47.843, 13.819, -19.551, -17.649]
  MoveL 1576 to (99.87, 1737.84, 513.19) mm, rotated rx 180 ry 0 rz -88.32 deg; joints [4.768, -21.524, -47.726, 13.754, -19.499, -17.558]
  MoveL 1577 to (99, 1740.55, 513.19) mm, rotated rx 180 ry 0 rz -88.32 deg; joints [4.722, -21.364, -47.608, 13.689, -19.447, -17.468]
  MoveL 1578 to (98.13, 1743.27, 513.19) mm, rotated rx 180 ry 0 rz -88.32 deg; joints [4.676, -21.203, -47.491, 13.624, -19.396, -17.378]
  MoveL 1579 to (97.27, 1745.98, 513.19) mm, rotated rx 180 ry 0 rz -88.32 deg; joints [4.63, -21.043, -47.373, 13.561, -19.345, -17.289]
  MoveL 1580 to (96.42, 1748.7, 513.19) mm, rotated rx -180 ry 0 rz -88.32 deg; joints [4.586, -20.883, -47.255, 13.497, -19.295, -17.201]
  MoveL 1581 to (95.57, 1751.43, 513.19) mm, rotated rx -180 ry 0 rz -88.32 deg; joints [4.541, -20.723, -47.136, 13.434, -19.245, -17.113]
  MoveL 1582 to (94.73, 1754.15, 513.19) mm, rotated rx -180 ry 0 rz -88.32 deg; joints [4.497, -20.563, -47.018, 13.372, -19.196, -17.026]
  MoveL 1583 to (93.9, 1756.88, 513.19) mm, rotated rx 180 ry 0 rz -88.32 deg; joints [4.454, -20.403, -46.899, 13.309, -19.147, -16.94]
  MoveL 1584 to (93.08, 1759.6, 513.19) mm, rotated rx -180 ry 0 rz -88.32 deg; joints [4.411, -20.243, -46.78, 13.248, -19.098, -16.855]
  MoveL 1585 to (92.27, 1762.34, 513.19) mm, rotated rx 180 ry 0 rz -88.32 deg; joints [4.369, -20.083, -46.66, 13.187, -19.05, -16.77]
  MoveL 1586 to (91.46, 1765.07, 513.19) mm, rotated rx 180 ry 0 rz -88.32 deg; joints [4.327, -19.924, -46.541, 13.126, -19.002, -16.686]
  MoveL 1587 to (90.66, 1767.8, 513.19) mm, rotated rx -180 ry 0 rz -88.32 deg; joints [4.285, -19.764, -46.421, 13.066, -18.955, -16.602]
  MoveL 1588 to (89.87, 1770.54, 513.19) mm, rotated rx -180 ry 0 rz -88.32 deg; joints [4.244, -19.605, -46.301, 13.006, -18.909, -16.52]
  MoveL 1589 to (89.08, 1773.28, 513.19) mm, rotated rx 180 ry 0 rz -88.32 deg; joints [4.204, -19.445, -46.181, 12.947, -18.862, -16.438]
  MoveL 1590 to (88.31, 1776.02, 513.19) mm, rotated rx -180 ry 0 rz -88.32 deg; joints [4.163, -19.286, -46.06, 12.888, -18.816, -16.357]
  MoveL 1591 to (87.54, 1778.77, 513.19) mm, rotated rx -180 ry 0 rz -88.32 deg; joints [4.124, -19.127, -45.94, 12.83, -18.771, -16.276]
  MoveL 1592 to (86.78, 1781.51, 513.19) mm, rotated rx -180 ry 0 rz -88.32 deg; joints [4.085, -18.968, -45.819, 12.772, -18.726, -16.197]
  MoveL 1593 to (86.02, 1784.26, 513.19) mm, rotated rx 180 ry 0 rz -88.32 deg; joints [4.046, -18.809, -45.698, 12.715, -18.681, -16.118]
  MoveL 1594 to (85.28, 1787.01, 513.19) mm, rotated rx 180 ry 0 rz -88.32 deg; joints [4.008, -18.65, -45.577, 12.658, -18.637, -16.039]
  MoveL 1595 to (84.54, 1789.77, 513.19) mm, rotated rx 180 ry 0 rz -88.32 deg; joints [3.97, -18.491, -45.455, 12.602, -18.593, -15.962]
  MoveL 1596 to (83.81, 1792.52, 513.19) mm, rotated rx -180 ry 0 rz -88.32 deg; joints [3.933, -18.332, -45.333, 12.546, -18.55, -15.885]
  MoveL 1597 to (83.09, 1795.28, 513.19) mm, rotated rx -180 ry 0 rz -88.32 deg; joints [3.896, -18.174, -45.211, 12.49, -18.507, -15.809]
  MoveL 1598 to (82.37, 1798.04, 513.19) mm, rotated rx 180 ry 0 rz -88.32 deg; joints [3.859, -18.015, -45.089, 12.436, -18.465, -15.734]
  MoveL 1599 to (81.67, 1800.8, 513.19) mm, rotated rx 180 ry 0 rz -88.32 deg; joints [3.823, -17.857, -44.967, 12.381, -18.423, -15.659]
  MoveL 1600 to (80.97, 1803.56, 513.19) mm, rotated rx 180 ry 0 rz -88.32 deg; joints [3.788, -17.699, -44.844, 12.327, -18.381, -15.585]
  MoveL 1601 to (80.28, 1806.33, 513.19) mm, rotated rx -180 ry 0 rz -88.32 deg; joints [3.752, -17.541, -44.721, 12.274, -18.34, -15.512]
  MoveL 1602 to (79.59, 1809.09, 513.19) mm, rotated rx -180 ry 0 rz -88.32 deg; joints [3.718, -17.382, -44.598, 12.221, -18.299, -15.44]
  MoveL 1603 to (78.92, 1811.86, 513.19) mm, rotated rx -180 ry 0 rz -88.32 deg; joints [3.684, -17.225, -44.475, 12.169, -18.259, -15.368]
  MoveL 1604 to (78.25, 1814.63, 513.19) mm, rotated rx 180 ry 0 rz -88.32 deg; joints [3.65, -17.067, -44.351, 12.117, -18.219, -15.298]
  MoveL 1605 to (77.59, 1817.4, 513.19) mm, rotated rx 180 ry 0 rz -88.32 deg; joints [3.616, -16.909, -44.228, 12.066, -18.18, -15.228]
  MoveL 1606 to (76.94, 1820.18, 513.19) mm, rotated rx 180 ry 0 rz -88.32 deg; joints [3.583, -16.752, -44.104, 12.015, -18.141, -15.158]
  MoveL 1607 to (76.29, 1822.95, 513.19) mm, rotated rx -180 ry 0 rz -88.32 deg; joints [3.551, -16.594, -43.98, 11.965, -18.102, -15.09]
  MoveL 1608 to (75.65, 1825.73, 513.19) mm, rotated rx -180 ry 0 rz -88.32 deg; joints [3.519, -16.437, -43.856, 11.915, -18.064, -15.022]
  MoveL 1609 to (75.03, 1828.51, 513.19) mm, rotated rx -180 ry 0 rz -88.32 deg; joints [3.487, -16.28, -43.731, 11.866, -18.026, -14.955]
  MoveL 1610 to (74.4, 1831.29, 513.19) mm, rotated rx -180 ry 0 rz -88.32 deg; joints [3.456, -16.123, -43.606, 11.818, -17.989, -14.889]
  MoveL 1611 to (73.79, 1834.07, 513.19) mm, rotated rx 180 ry 0 rz -88.32 deg; joints [3.425, -15.966, -43.482, 11.77, -17.952, -14.823]
  MoveL 1612 to (73.18, 1836.86, 513.19) mm, rotated rx -180 ry 0 rz -88.32 deg; joints [3.395, -15.809, -43.356, 11.722, -17.915, -14.758]
  MoveL 1613 to (72.59, 1839.65, 513.19) mm, rotated rx 180 ry 0 rz -88.32 deg; joints [3.365, -15.652, -43.231, 11.675, -17.879, -14.695]
  MoveL 1614 to (72, 1842.43, 513.19) mm, rotated rx -180 ry 0 rz -88.32 deg; joints [3.335, -15.496, -43.106, 11.629, -17.843, -14.631]
  MoveL 1615 to (71.41, 1845.22, 513.19) mm, rotated rx -180 ry 0 rz -88.32 deg; joints [3.306, -15.339, -42.98, 11.583, -17.808, -14.569]
  MoveL 1616 to (70.84, 1848.02, 513.19) mm, rotated rx 180 ry 0 rz -88.32 deg; joints [3.277, -15.183, -42.854, 11.537, -17.773, -14.507]
  MoveL 1617 to (70.27, 1850.81, 513.19) mm, rotated rx 180 ry 0 rz -88.32 deg; joints [3.249, -15.027, -42.728, 11.493, -17.739, -14.446]
  MoveL 1618 to (69.71, 1853.6, 513.19) mm, rotated rx 180 ry 0 rz -88.32 deg; joints [3.221, -14.871, -42.602, 11.448, -17.705, -14.386]
  MoveL 1619 to (69.16, 1856.4, 513.19) mm, rotated rx 180 ry 0 rz -88.32 deg; joints [3.193, -14.715, -42.476, 11.404, -17.671, -14.327]
  MoveL 1620 to (68.62, 1859.2, 513.19) mm, rotated rx 180 ry 0 rz -88.32 deg; joints [3.166, -14.559, -42.349, 11.361, -17.638, -14.268]
  MoveL 1621 to (68.09, 1862, 513.19) mm, rotated rx 180 ry 0 rz -88.32 deg; joints [3.14, -14.404, -42.222, 11.319, -17.605, -14.21]
  MoveL 1622 to (67.56, 1864.8, 513.19) mm, rotated rx -180 ry 0 rz -88.32 deg; joints [3.113, -14.248, -42.095, 11.277, -17.572, -14.153]
  MoveL 1623 to (67.04, 1867.6, 513.19) mm, rotated rx 180 ry 0 rz -88.32 deg; joints [3.087, -14.093, -41.968, 11.235, -17.54, -14.097]
  MoveL 1624 to (66.53, 1870.4, 513.19) mm, rotated rx -180 ry 0 rz -88.32 deg; joints [3.062, -13.938, -41.841, 11.194, -17.508, -14.042]
  MoveL 1625 to (66.02, 1873.21, 513.19) mm, rotated rx 180 ry 0 rz -88.32 deg; joints [3.037, -13.783, -41.713, 11.154, -17.477, -13.987]
  MoveL 1626 to (65.53, 1876.01, 513.19) mm, rotated rx -180 ry 0 rz -88.32 deg; joints [3.012, -13.628, -41.585, 11.114, -17.446, -13.933]
  MoveL 1627 to (65.04, 1878.82, 513.19) mm, rotated rx -180 ry 0 rz -88.32 deg; joints [2.988, -13.473, -41.458, 11.074, -17.416, -13.88]
  MoveL 1628 to (64.56, 1881.63, 513.19) mm, rotated rx -180 ry 0 rz -88.32 deg; joints [2.964, -13.318, -41.329, 11.036, -17.386, -13.827]
  MoveL 1629 to (64.09, 1884.44, 513.19) mm, rotated rx -180 ry 0 rz -88.32 deg; joints [2.94, -13.164, -41.201, 10.998, -17.356, -13.776]
  MoveL 1630 to (63.62, 1887.25, 513.19) mm, rotated rx 180 ry 0 rz -88.32 deg; joints [2.917, -13.01, -41.073, 10.96, -17.327, -13.725]
  MoveL 1631 to (63.17, 1890.07, 513.19) mm, rotated rx -180 ry 0 rz -88.32 deg; joints [2.894, -12.855, -40.944, 10.923, -17.298, -13.675]
  MoveL 1632 to (62.72, 1892.88, 513.19) mm, rotated rx -180 ry 0 rz -88.32 deg; joints [2.872, -12.701, -40.815, 10.886, -17.269, -13.626]
  MoveL 1633 to (62.28, 1895.7, 513.19) mm, rotated rx 180 ry 0 rz -88.32 deg; joints [2.85, -12.547, -40.686, 10.851, -17.241, -13.577]
  MoveL 1634 to (61.84, 1898.51, 513.19) mm, rotated rx -180 ry 0 rz -88.32 deg; joints [2.828, -12.394, -40.557, 10.815, -17.213, -13.53]
  MoveL 1635 to (61.42, 1901.33, 513.19) mm, rotated rx -180 ry 0 rz -88.32 deg; joints [2.807, -12.24, -40.428, 10.78, -17.186, -13.483]
  MoveL 1636 to (61, 1904.15, 513.19) mm, rotated rx -180 ry 0 rz -88.32 deg; joints [2.786, -12.087, -40.299, 10.746, -17.159, -13.437]
  MoveL 1637 to (60.59, 1906.97, 513.19) mm, rotated rx 180 ry 0 rz -88.32 deg; joints [2.765, -11.933, -40.169, 10.713, -17.132, -13.391]
  MoveL 1638 to (60.19, 1909.79, 513.19) mm, rotated rx -180 ry 0 rz -88.32 deg; joints [2.745, -11.78, -40.039, 10.68, -17.106, -13.347]
  MoveL 1639 to (59.8, 1912.61, 513.19) mm, rotated rx -180 ry 0 rz -88.32 deg; joints [2.725, -11.627, -39.909, 10.647, -17.08, -13.303]
  MoveL 1640 to (59.41, 1915.44, 513.19) mm, rotated rx 180 ry 0 rz -88.32 deg; joints [2.706, -11.474, -39.779, 10.615, -17.054, -13.26]
  MoveL 1641 to (59.03, 1918.26, 513.19) mm, rotated rx 180 ry 0 rz -88.32 deg; joints [2.687, -11.322, -39.649, 10.584, -17.029, -13.218]
  MoveL 1642 to (58.67, 1921.09, 513.19) mm, rotated rx -180 ry 0 rz -88.32 deg; joints [2.668, -11.169, -39.518, 10.553, -17.005, -13.176]
  MoveL 1643 to (58.3, 1923.91, 513.19) mm, rotated rx 180 ry 0 rz -88.32 deg; joints [2.65, -11.017, -39.388, 10.523, -16.98, -13.136]
  MoveL 1644 to (57.95, 1926.74, 513.19) mm, rotated rx 180 ry 0 rz -88.32 deg; joints [2.632, -10.864, -39.257, 10.493, -16.956, -13.096]
  MoveL 1645 to (57.6, 1929.57, 513.19) mm, rotated rx -180 ry 0 rz -88.32 deg; joints [2.614, -10.712, -39.126, 10.464, -16.933, -13.057]
  MoveL 1646 to (57.27, 1932.4, 513.19) mm, rotated rx 180 ry 0 rz -88.32 deg; joints [2.597, -10.56, -38.995, 10.436, -16.909, -13.018]
  MoveL 1647 to (56.94, 1935.23, 513.19) mm, rotated rx 180 ry 0 rz -88.32 deg; joints [2.58, -10.408, -38.864, 10.408, -16.886, -12.981]
  MoveL 1648 to (56.61, 1938.06, 513.19) mm, rotated rx -180 ry 0 rz -88.32 deg; joints [2.564, -10.257, -38.732, 10.381, -16.864, -12.944]
  MoveL 1649 to (56.3, 1940.9, 513.19) mm, rotated rx -180 ry 0 rz -88.32 deg; joints [2.547, -10.105, -38.601, 10.354, -16.842, -12.908]
  MoveL 1650 to (55.99, 1943.73, 513.19) mm, rotated rx 180 ry 0 rz -88.32 deg; joints [2.531, -9.954, -38.469, 10.328, -16.82, -12.873]
  MoveL 1651 to (55.7, 1946.56, 513.19) mm, rotated rx -180 ry 0 rz -88.32 deg; joints [2.516, -9.803, -38.337, 10.302, -16.799, -12.838]
  MoveL 1652 to (55.41, 1949.4, 513.19) mm, rotated rx 180 ry 0 rz -88.32 deg; joints [2.501, -9.652, -38.205, 10.277, -16.777, -12.805]
  MoveL 1653 to (55.12, 1952.23, 513.19) mm, rotated rx -180 ry 0 rz -88.32 deg; joints [2.486, -9.501, -38.073, 10.253, -16.757, -12.772]
  MoveL 1654 to (54.85, 1955.07, 513.19) mm, rotated rx -180 ry 0 rz -88.32 deg; joints [2.471, -9.35, -37.94, 10.229, -16.736, -12.74]
  MoveL 1655 to (54.58, 1957.91, 513.19) mm, rotated rx -180 ry 0 rz -88.32 deg; joints [2.457, -9.2, -37.808, 10.206, -16.716, -12.708]
  MoveL 1656 to (54.33, 1960.75, 513.19) mm, rotated rx 180 ry 0 rz -88.32 deg; joints [2.444, -9.049, -37.675, 10.183, -16.697, -12.678]
  MoveL 1657 to (54.07, 1963.59, 513.19) mm, rotated rx 180 ry 0 rz -88.32 deg; joints [2.43, -8.899, -37.542, 10.161, -16.678, -12.648]
  MoveL 1658 to (53.83, 1966.43, 513.19) mm, rotated rx -180 ry 0 rz -88.32 deg; joints [2.417, -8.749, -37.409, 10.14, -16.659, -12.619]
  MoveL 1659 to (53.6, 1969.27, 513.19) mm, rotated rx 180 ry 0 rz -88.32 deg; joints [2.404, -8.599, -37.276, 10.119, -16.64, -12.591]
  MoveL 1660 to (53.37, 1972.11, 513.19) mm, rotated rx 180 ry 0 rz -88.32 deg; joints [2.392, -8.449, -37.143, 10.098, -16.622, -12.563]
  MoveL 1661 to (53.15, 1974.95, 513.19) mm, rotated rx 180 ry 0 rz -88.32 deg; joints [2.38, -8.299, -37.01, 10.079, -16.604, -12.536]
  MoveL 1662 to (52.94, 1977.79, 513.19) mm, rotated rx 180 ry 0 rz -88.32 deg; joints [2.368, -8.15, -36.876, 10.059, -16.587, -12.51]
  MoveL 1663 to (52.74, 1980.63, 513.19) mm, rotated rx 180 ry 0 rz -88.32 deg; joints [2.356, -8.001, -36.742, 10.041, -16.569, -12.485]
  MoveL 1664 to (52.55, 1983.48, 513.19) mm, rotated rx 180 ry 0 rz -88.32 deg; joints [2.345, -7.851, -36.608, 10.023, -16.553, -12.461]
  MoveL 1665 to (52.36, 1986.32, 513.19) mm, rotated rx 180 ry 0 rz -88.32 deg; joints [2.334, -7.702, -36.474, 10.005, -16.536, -12.437]
  MoveL 1666 to (52.18, 1989.16, 513.19) mm, rotated rx -180 ry 0 rz -88.32 deg; joints [2.324, -7.554, -36.34, 9.988, -16.52, -12.414]
  MoveL 1667 to (52.01, 1992.01, 513.19) mm, rotated rx -180 ry 0 rz -88.32 deg; joints [2.314, -7.405, -36.206, 9.972, -16.504, -12.392]
  MoveL 1668 to (51.85, 1994.85, 513.19) mm, rotated rx 180 ry 0 rz -88.32 deg; joints [2.304, -7.256, -36.072, 9.956, -16.489, -12.371]
  MoveL 1669 to (51.69, 1997.7, 513.19) mm, rotated rx 180 ry 0 rz -88.32 deg; joints [2.294, -7.108, -35.937, 9.941, -16.474, -12.35]
  MoveL 1670 to (51.55, 2000.55, 513.19) mm, rotated rx 180 ry 0 rz -88.32 deg; joints [2.285, -6.96, -35.802, 9.926, -16.459, -12.33]
  MoveL 1671 to (51.41, 2003.39, 513.19) mm, rotated rx -180 ry 0 rz -88.32 deg; joints [2.276, -6.812, -35.668, 9.912, -16.445, -12.311]
  MoveL 1672 to (51.28, 2006.24, 513.19) mm, rotated rx 180 ry 0 rz -88.32 deg; joints [2.267, -6.664, -35.533, 9.899, -16.431, -12.293]
  MoveL 1673 to (51.15, 2009.09, 513.19) mm, rotated rx 180 ry 0 rz -88.32 deg; joints [2.259, -6.516, -35.398, 9.886, -16.417, -12.275]
  MoveL 1674 to (51.04, 2011.93, 513.19) mm, rotated rx 180 ry 0 rz -88.32 deg; joints [2.251, -6.368, -35.262, 9.874, -16.404, -12.258]
  MoveL 1675 to (50.93, 2014.78, 513.19) mm, rotated rx -180 ry 0 rz -88.32 deg; joints [2.243, -6.221, -35.127, 9.862, -16.391, -12.242]
  MoveL 1676 to (50.83, 2017.63, 513.19) mm, rotated rx 180 ry 0 rz -88.32 deg; joints [2.236, -6.074, -34.991, 9.851, -16.378, -12.227]
  MoveL 1677 to (50.74, 2020.48, 513.19) mm, rotated rx 180 ry 0 rz -88.32 deg; joints [2.229, -5.927, -34.856, 9.84, -16.366, -12.212]
  MoveL 1678 to (50.66, 2023.33, 513.19) mm, rotated rx 180 ry 0 rz -88.32 deg; joints [2.222, -5.78, -34.72, 9.83, -16.354, -12.198]
  MoveL 1679 to (50.58, 2026.18, 513.19) mm, rotated rx 180 ry 0 rz -88.32 deg; joints [2.216, -5.633, -34.584, 9.82, -16.342, -12.185]
  MoveL 1680 to (50.52, 2029.02, 513.19) mm, rotated rx -180 ry 0 rz -88.32 deg; joints [2.21, -5.486, -34.448, 9.811, -16.331, -12.172]
  MoveL 1681 to (50.46, 2031.87, 513.19) mm, rotated rx -180 ry 0 rz -88.32 deg; joints [2.204, -5.34, -34.312, 9.803, -16.319, -12.161]
  MoveL 1682 to (50.41, 2034.72, 513.19) mm, rotated rx 180 ry 0 rz -88.32 deg; joints [2.198, -5.193, -34.176, 9.795, -16.309, -12.15]
  MoveL 1683 to (50.37, 2037.57, 513.19) mm, rotated rx -180 ry 0 rz -88.32 deg; joints [2.193, -5.047, -34.039, 9.788, -16.298, -12.139]
  MoveL 1684 to (50.33, 2040.42, 513.19) mm, rotated rx -180 ry 0 rz -88.32 deg; joints [2.188, -4.901, -33.903, 9.781, -16.288, -12.13]
  MoveL 1685 to (50.3, 2043.27, 513.19) mm, rotated rx -180 ry 0 rz -88.32 deg; joints [2.183, -4.755, -33.766, 9.775, -16.279, -12.121]
  MoveL 1686 to (50.28, 2046.12, 513.19) mm, rotated rx 180 ry 0 rz -88.32 deg; joints [2.179, -4.61, -33.629, 9.769, -16.269, -12.113]
  MoveL 1687 to (50.27, 2048.97, 513.19) mm, rotated rx -180 ry 0 rz -88.32 deg; joints [2.175, -4.464, -33.492, 9.764, -16.26, -12.105]
  MoveL 1688 to (50.27, 2051.82, 513.19) mm, rotated rx -180 ry 0 rz -88.32 deg; joints [2.171, -4.319, -33.355, 9.759, -16.251, -12.099]
  MoveL 1689 to (50.28, 2054.67, 513.19) mm, rotated rx -180 ry 0 rz -88.32 deg; joints [2.167, -4.174, -33.218, 9.755, -16.243, -12.093]
  MoveL 1690 to (50.29, 2057.52, 513.19) mm, rotated rx -180 ry 0 rz -88.32 deg; joints [2.164, -4.028, -33.08, 9.752, -16.235, -12.087]
  MoveL 1691 to (50.31, 2060.37, 513.19) mm, rotated rx 180 ry 0 rz -88.32 deg; joints [2.161, -3.884, -32.943, 9.749, -16.227, -12.083]
  MoveL 1692 to (50.34, 2063.22, 513.19) mm, rotated rx 180 ry 0 rz -88.32 deg; joints [2.158, -3.739, -32.805, 9.746, -16.22, -12.079]
  MoveL 1693 to (50.38, 2066.07, 513.19) mm, rotated rx 180 ry 0 rz -88.32 deg; joints [2.156, -3.594, -32.668, 9.744, -16.212, -12.076]
  MoveL 1694 to (50.42, 2068.92, 513.19) mm, rotated rx 180 ry 0 rz -88.32 deg; joints [2.154, -3.45, -32.53, 9.743, -16.206, -12.073]
  MoveL 1695 to (50.47, 2071.77, 513.19) mm, rotated rx -180 ry 0 rz -88.32 deg; joints [2.152, -3.306, -32.392, 9.742, -16.199, -12.071]
  MoveL 1696 to (50.54, 2074.62, 513.19) mm, rotated rx 180 ry 0 rz -88.32 deg; joints [2.151, -3.161, -32.254, 9.742, -16.193, -12.07]
  MoveL 1697 to (50.6, 2077.47, 513.19) mm, rotated rx -180 ry 0 rz -88.32 deg; joints [2.149, -3.017, -32.116, 9.742, -16.187, -12.07]
  MoveL 1698 to (50.68, 2080.32, 513.19) mm, rotated rx -180 ry 0 rz -88.32 deg; joints [2.148, -2.874, -31.978, 9.743, -16.181, -12.07]
  MoveL 1699 to (50.77, 2083.16, 513.19) mm, rotated rx 180 ry 0 rz -88.32 deg; joints [2.148, -2.73, -31.839, 9.744, -16.176, -12.071]
  MoveL 1700 to (50.86, 2086.01, 513.19) mm, rotated rx -180 ry 0 rz -88.32 deg; joints [2.147, -2.587, -31.701, 9.746, -16.171, -12.072]
  MoveL 1701 to (50.96, 2088.86, 513.19) mm, rotated rx -180 ry 0 rz -88.32 deg; joints [2.147, -2.443, -31.562, 9.748, -16.166, -12.075]
  MoveL 1702 to (51.07, 2091.71, 513.19) mm, rotated rx -180 ry 0 rz -88.32 deg; joints [2.147, -2.3, -31.423, 9.751, -16.162, -12.078]
  MoveL 1703 to (51.19, 2094.56, 513.19) mm, rotated rx -180 ry 0 rz -88.32 deg; joints [2.147, -2.157, -31.284, 9.754, -16.158, -12.081]
  MoveL 1704 to (51.31, 2097.4, 513.19) mm, rotated rx 180 ry 0 rz -88.32 deg; joints [2.148, -2.014, -31.145, 9.758, -16.154, -12.085]
  MoveL 1705 to (51.44, 2100.25, 513.19) mm, rotated rx -180 ry 0 rz -88.32 deg; joints [2.149, -1.871, -31.006, 9.762, -16.151, -12.09]
  MoveL 1706 to (51.59, 2103.1, 513.19) mm, rotated rx 180 ry 0 rz -88.32 deg; joints [2.15, -1.729, -30.867, 9.767, -16.148, -12.096]
  MoveL 1707 to (51.73, 2105.94, 513.19) mm, rotated rx -180 ry 0 rz -88.32 deg; joints [2.151, -1.586, -30.728, 9.772, -16.145, -12.102]
  MoveL 1708 to (51.89, 2108.79, 513.19) mm, rotated rx -180 ry 0 rz -88.32 deg; joints [2.153, -1.444, -30.588, 9.778, -16.142, -12.109]
  MoveL 1709 to (52.06, 2111.63, 513.19) mm, rotated rx 180 ry 0 rz -88.32 deg; joints [2.155, -1.302, -30.449, 9.784, -16.14, -12.116]
  MoveL 1710 to (52.23, 2114.48, 513.19) mm, rotated rx 180 ry 0 rz -88.32 deg; joints [2.157, -1.16, -30.309, 9.791, -16.138, -12.125]
  MoveL 1711 to (52.41, 2117.32, 513.19) mm, rotated rx 180 ry 0 rz -88.32 deg; joints [2.159, -1.018, -30.169, 9.798, -16.137, -12.133]
  MoveL 1712 to (52.6, 2120.17, 513.19) mm, rotated rx -180 ry 0 rz -88.32 deg; joints [2.162, -0.877, -30.029, 9.806, -16.135, -12.143]
  MoveL 1713 to (52.8, 2123.01, 513.19) mm, rotated rx -180 ry 0 rz -88.32 deg; joints [2.165, -0.735, -29.889, 9.814, -16.134, -12.153]
  MoveL 1714 to (53, 2125.85, 513.19) mm, rotated rx 180 ry 0 rz -88.32 deg; joints [2.168, -0.594, -29.749, 9.823, -16.134, -12.163]
  MoveL 1715 to (53.21, 2128.69, 513.19) mm, rotated rx 180 ry 0 rz -88.32 deg; joints [2.172, -0.453, -29.609, 9.832, -16.133, -12.175]
  MoveL 1716 to (53.43, 2131.53, 513.19) mm, rotated rx -180 ry 0 rz -88.32 deg; joints [2.175, -0.312, -29.469, 9.842, -16.133, -12.187]
  MoveL 1717 to (53.66, 2134.37, 513.19) mm, rotated rx -180 ry 0 rz -88.32 deg; joints [2.179, -0.171, -29.328, 9.852, -16.133, -12.199]
  MoveL 1718 to (53.9, 2137.22, 513.19) mm, rotated rx 180 ry 0 rz -88.32 deg; joints [2.184, -0.03, -29.188, 9.862, -16.134, -12.212]
  MoveL 1719 to (54.14, 2140.05, 513.19) mm, rotated rx 180 ry 0 rz -88.32 deg; joints [2.188, 0.11, -29.047, 9.873, -16.134, -12.226]
  MoveL 1720 to (54.4, 2142.89, 513.19) mm, rotated rx -180 ry 0 rz -88.32 deg; joints [2.193, 0.251, -28.906, 9.885, -16.135, -12.24]
  MoveL 1721 to (54.66, 2145.73, 513.19) mm, rotated rx 180 ry 0 rz -88.32 deg; joints [2.198, 0.391, -28.766, 9.897, -16.137, -12.255]
  MoveL 1722 to (54.93, 2148.57, 513.19) mm, rotated rx -180 ry 0 rz -88.32 deg; joints [2.203, 0.531, -28.625, 9.909, -16.138, -12.271]
  MoveL 1723 to (55.2, 2151.4, 513.19) mm, rotated rx 180 ry 0 rz -88.32 deg; joints [2.208, 0.671, -28.484, 9.922, -16.14, -12.287]
  MoveL 1724 to (55.49, 2154.24, 513.19) mm, rotated rx 180 ry 0 rz -88.32 deg; joints [2.214, 0.811, -28.342, 9.935, -16.142, -12.304]
  MoveL 1725 to (55.78, 2157.07, 513.19) mm, rotated rx -180 ry 0 rz -88.32 deg; joints [2.22, 0.951, -28.201, 9.949, -16.145, -12.321]
  MoveL 1726 to (56.08, 2159.91, 513.19) mm, rotated rx 180 ry 0 rz -88.32 deg; joints [2.226, 1.09, -28.06, 9.963, -16.148, -12.339]
  MoveL 1727 to (56.39, 2162.74, 513.19) mm, rotated rx 180 ry 0 rz -88.32 deg; joints [2.232, 1.23, -27.918, 9.978, -16.151, -12.357]
  MoveL 1728 to (56.7, 2165.57, 513.19) mm, rotated rx 180 ry 0 rz -88.32 deg; joints [2.239, 1.369, -27.777, 9.993, -16.154, -12.376]
  MoveL 1729 to (57.03, 2168.41, 513.19) mm, rotated rx -180 ry 0 rz -88.32 deg; joints [2.246, 1.508, -27.635, 10.008, -16.158, -12.396]
  MoveL 1730 to (57.36, 2171.24, 513.19) mm, rotated rx -180 ry 0 rz -88.32 deg; joints [2.253, 1.647, -27.493, 10.024, -16.161, -12.416]
  MoveL 1731 to (57.7, 2174.07, 513.19) mm, rotated rx 180 ry 0 rz -88.32 deg; joints [2.26, 1.785, -27.351, 10.04, -16.166, -12.436]
  MoveL 1732 to (58.05, 2176.89, 513.19) mm, rotated rx 180 ry 0 rz -88.32 deg; joints [2.268, 1.924, -27.209, 10.057, -16.17, -12.458]
  MoveL 1733 to (58.4, 2179.72, 513.19) mm, rotated rx -180 ry 0 rz -88.32 deg; joints [2.276, 2.063, -27.067, 10.074, -16.175, -12.479]
  MoveL 1734 to (58.77, 2182.55, 513.19) mm, rotated rx 180 ry 0 rz -88.32 deg; joints [2.284, 2.201, -26.925, 10.092, -16.18, -12.502]
  MoveL 1735 to (59.14, 2185.37, 513.19) mm, rotated rx 180 ry 0 rz -88.32 deg; joints [2.292, 2.339, -26.783, 10.11, -16.185, -12.525]
  MoveL 1736 to (59.52, 2188.2, 513.19) mm, rotated rx -180 ry 0 rz -88.32 deg; joints [2.3, 2.477, -26.641, 10.128, -16.191, -12.548]
  MoveL 1737 to (59.91, 2191.02, 513.19) mm, rotated rx -180 ry 0 rz -88.32 deg; joints [2.309, 2.615, -26.498, 10.147, -16.197, -12.572]
  MoveL 1738 to (60.3, 2193.84, 513.19) mm, rotated rx 180 ry 0 rz -88.32 deg; joints [2.318, 2.753, -26.356, 10.166, -16.203, -12.596]
  MoveL 1739 to (60.71, 2196.67, 513.19) mm, rotated rx 180 ry 0 rz -88.32 deg; joints [2.327, 2.89, -26.213, 10.185, -16.209, -12.621]
  MoveL 1740 to (61.12, 2199.49, 513.19) mm, rotated rx 180 ry 0 rz -88.32 deg; joints [2.336, 3.028, -26.07, 10.205, -16.216, -12.647]
  MoveL 1741 to (61.54, 2202.3, 513.19) mm, rotated rx -180 ry 0 rz -88.32 deg; joints [2.346, 3.165, -25.927, 10.226, -16.223, -12.673]
  MoveL 1742 to (61.96, 2205.12, 513.19) mm, rotated rx 180 ry 0 rz -88.32 deg; joints [2.356, 3.302, -25.785, 10.246, -16.23, -12.699]
  MoveL 1743 to (62.4, 2207.94, 513.19) mm, rotated rx 180 ry 0 rz -88.32 deg; joints [2.366, 3.439, -25.642, 10.267, -16.237, -12.726]
  MoveL 1744 to (62.84, 2210.75, 513.19) mm, rotated rx 180 ry 0 rz -88.32 deg; joints [2.376, 3.576, -25.498, 10.289, -16.245, -12.754]
  MoveL 1745 to (63.29, 2213.57, 513.19) mm, rotated rx -180 ry 0 rz -88.32 deg; joints [2.387, 3.713, -25.355, 10.31, -16.253, -12.782]
  MoveL 1746 to (63.75, 2216.38, 513.19) mm, rotated rx -180 ry 0 rz -88.32 deg; joints [2.397, 3.849, -25.212, 10.333, -16.261, -12.81]
  MoveL 1747 to (64.22, 2219.19, 513.19) mm, rotated rx -180 ry 0 rz -88.32 deg; joints [2.408, 3.986, -25.069, 10.355, -16.27, -12.839]
  MoveL 1748 to (64.69, 2222, 513.19) mm, rotated rx 180 ry 0 rz -88.32 deg; joints [2.419, 4.122, -24.925, 10.378, -16.279, -12.869]
  MoveL 1749 to (65.18, 2224.81, 513.19) mm, rotated rx 180 ry 0 rz -88.32 deg; joints [2.431, 4.258, -24.782, 10.401, -16.288, -12.899]
  MoveL 1750 to (65.67, 2227.62, 513.19) mm, rotated rx -180 ry 0 rz -88.32 deg; joints [2.442, 4.394, -24.638, 10.425, -16.297, -12.929]
  MoveL 1751 to (66.16, 2230.42, 513.19) mm, rotated rx -180 ry 0 rz -88.32 deg; joints [2.454, 4.53, -24.494, 10.449, -16.307, -12.96]
  MoveL 1752 to (66.67, 2233.23, 513.19) mm, rotated rx 180 ry 0 rz -88.32 deg; joints [2.466, 4.666, -24.35, 10.473, -16.317, -12.991]
  MoveL 1753 to (67.18, 2236.03, 513.19) mm, rotated rx -180 ry 0 rz -88.32 deg; joints [2.478, 4.801, -24.206, 10.498, -16.327, -13.023]
  MoveL 1754 to (67.71, 2238.83, 513.19) mm, rotated rx -180 ry 0 rz -88.32 deg; joints [2.49, 4.937, -24.062, 10.523, -16.337, -13.055]
  MoveL 1755 to (68.24, 2241.63, 513.19) mm, rotated rx 180 ry 0 rz -88.32 deg; joints [2.503, 5.072, -23.918, 10.548, -16.348, -13.088]
  MoveL 1756 to (68.77, 2244.43, 513.19) mm, rotated rx 180 ry 0 rz -88.32 deg; joints [2.516, 5.207, -23.774, 10.574, -16.359, -13.121]
  MoveL 1757 to (69.32, 2247.23, 513.19) mm, rotated rx 180 ry 0 rz -88.32 deg; joints [2.529, 5.342, -23.63, 10.599, -16.37, -13.155]
  MoveL 1758 to (69.87, 2250.02, 513.19) mm, rotated rx 180 ry 0 rz -88.32 deg; joints [2.542, 5.477, -23.485, 10.626, -16.381, -13.189]
  MoveL 1759 to (70.43, 2252.82, 513.19) mm, rotated rx -180 ry 0 rz -88.32 deg; joints [2.555, 5.612, -23.341, 10.652, -16.393, -13.223]
  MoveL 1760 to (71, 2255.61, 513.19) mm, rotated rx -180 ry 0 rz -88.32 deg; joints [2.569, 5.746, -23.196, 10.679, -16.405, -13.258]
  MoveL 1761 to (71.58, 2258.4, 513.19) mm, rotated rx -180 ry 0 rz -88.32 deg; joints [2.583, 5.881, -23.052, 10.706, -16.417, -13.293]
  MoveL 1762 to (72.16, 2261.19, 513.19) mm, rotated rx -180 ry 0 rz -88.32 deg; joints [2.597, 6.015, -22.907, 10.734, -16.43, -13.329]
  MoveL 1763 to (72.75, 2263.98, 513.19) mm, rotated rx -180 ry 0 rz -88.32 deg; joints [2.611, 6.149, -22.762, 10.762, -16.443, -13.365]
  MoveL 1764 to (73.35, 2266.77, 513.19) mm, rotated rx -180 ry 0 rz -88.32 deg; joints [2.625, 6.283, -22.618, 10.79, -16.456, -13.402]
  MoveL 1765 to (73.96, 2269.55, 513.19) mm, rotated rx -180 ry 0 rz -88.32 deg; joints [2.64, 6.417, -22.473, 10.818, -16.469, -13.439]
  MoveL 1766 to (74.58, 2272.33, 513.19) mm, rotated rx -180 ry 0 rz -88.32 deg; joints [2.654, 6.551, -22.328, 10.847, -16.482, -13.476]
  MoveL 1767 to (75.2, 2275.11, 513.19) mm, rotated rx 180 ry 0 rz -88.32 deg; joints [2.669, 6.685, -22.182, 10.876, -16.496, -13.514]
  MoveL 1768 to (75.83, 2277.89, 513.19) mm, rotated rx -180 ry 0 rz -88.32 deg; joints [2.685, 6.818, -22.037, 10.905, -16.51, -13.552]
  MoveL 1769 to (76.47, 2280.67, 513.19) mm, rotated rx 180 ry 0 rz -88.32 deg; joints [2.7, 6.951, -21.892, 10.934, -16.524, -13.59]
  MoveL 1770 to (77.12, 2283.44, 513.19) mm, rotated rx 180 ry 0 rz -88.32 deg; joints [2.715, 7.085, -21.747, 10.964, -16.539, -13.629]
  MoveL 1771 to (77.77, 2286.22, 513.19) mm, rotated rx -180 ry 0 rz -88.32 deg; joints [2.731, 7.218, -21.601, 10.994, -16.554, -13.668]
  MoveL 1772 to (78.44, 2288.99, 513.19) mm, rotated rx -180 ry 0 rz -88.32 deg; joints [2.747, 7.351, -21.456, 11.025, -16.569, -13.708]
  MoveL 1773 to (79.11, 2291.76, 513.19) mm, rotated rx 180 ry 0 rz -88.32 deg; joints [2.763, 7.484, -21.31, 11.055, -16.584, -13.748]
  MoveL 1774 to (79.78, 2294.53, 513.19) mm, rotated rx 180 ry 0 rz -88.32 deg; joints [2.78, 7.616, -21.164, 11.086, -16.599, -13.789]
  MoveL 1775 to (80.47, 2297.29, 513.19) mm, rotated rx -180 ry 0 rz -88.32 deg; joints [2.796, 7.749, -21.019, 11.117, -16.615, -13.829]
  MoveL 1776 to (81.16, 2300.06, 513.19) mm, rotated rx -180 ry 0 rz -88.32 deg; joints [2.813, 7.881, -20.873, 11.149, -16.631, -13.87]
  MoveL 1777 to (81.87, 2302.82, 513.19) mm, rotated rx 180 ry 0 rz -88.32 deg; joints [2.83, 8.014, -20.727, 11.18, -16.647, -13.912]
  MoveL 1778 to (82.57, 2305.58, 513.19) mm, rotated rx 180 ry 0 rz -88.32 deg; joints [2.847, 8.146, -20.581, 11.212, -16.664, -13.954]
  MoveL 1779 to (83.29, 2308.34, 513.19) mm, rotated rx -180 ry 0 rz -88.32 deg; joints [2.864, 8.278, -20.435, 11.244, -16.68, -13.996]
  MoveL 1780 to (84.02, 2311.1, 513.19) mm, rotated rx 180 ry 0 rz -88.32 deg; joints [2.881, 8.41, -20.289, 11.276, -16.697, -14.038]
  MoveL 1781 to (84.75, 2313.85, 513.19) mm, rotated rx 180 ry 0 rz -88.32 deg; joints [2.899, 8.541, -20.142, 11.309, -16.715, -14.081]
  MoveL 1782 to (85.49, 2316.6, 513.19) mm, rotated rx -180 ry 0 rz -88.32 deg; joints [2.917, 8.673, -19.996, 11.342, -16.732, -14.124]
  MoveL 1783 to (86.24, 2319.35, 513.19) mm, rotated rx 180 ry 0 rz -88.32 deg; joints [2.935, 8.805, -19.85, 11.375, -16.75, -14.168]
  MoveL 1784 to (86.99, 2322.1, 513.19) mm, rotated rx 180 ry 0 rz -88.32 deg; joints [2.953, 8.936, -19.703, 11.408, -16.768, -14.211]
  MoveL 1785 to (87.75, 2324.85, 513.19) mm, rotated rx -180 ry 0 rz -88.32 deg; joints [2.971, 9.067, -19.557, 11.441, -16.786, -14.256]
  MoveL 1786 to (88.53, 2327.59, 513.19) mm, rotated rx 180 ry 0 rz -88.32 deg; joints [2.99, 9.198, -19.41, 11.475, -16.804, -14.3]
  MoveL 1787 to (89.3, 2330.33, 513.19) mm, rotated rx 180 ry 0 rz -88.32 deg; joints [3.008, 9.329, -19.263, 11.509, -16.823, -14.345]
  MoveL 1788 to (90.09, 2333.07, 513.19) mm, rotated rx 180 ry 0 rz -88.32 deg; joints [3.027, 9.46, -19.117, 11.543, -16.842, -14.39]
  MoveL 1789 to (90.88, 2335.81, 513.19) mm, rotated rx -180 ry 0 rz -88.32 deg; joints [3.046, 9.591, -18.97, 11.577, -16.861, -14.435]
  MoveL 1790 to (91.69, 2338.54, 513.19) mm, rotated rx -180 ry 0 rz -88.32 deg; joints [3.065, 9.721, -18.823, 11.612, -16.88, -14.481]
  MoveL 1791 to (92.49, 2341.27, 513.19) mm, rotated rx 180 ry 0 rz -88.32 deg; joints [3.085, 9.852, -18.676, 11.647, -16.9, -14.527]
  MoveL 1792 to (93.31, 2344, 513.19) mm, rotated rx 180 ry 0 rz -88.32 deg; joints [3.104, 9.982, -18.529, 11.681, -16.92, -14.573]
  MoveL 1793 to (94.14, 2346.73, 513.19) mm, rotated rx -180 ry 0 rz -88.32 deg; joints [3.124, 10.113, -18.382, 11.717, -16.94, -14.619]
  MoveL 1794 to (94.97, 2349.46, 513.19) mm, rotated rx -180 ry 0 rz -88.32 deg; joints [3.144, 10.243, -18.235, 11.752, -16.96, -14.666]
  MoveL 1795 to (95.81, 2352.18, 513.19) mm, rotated rx 180 ry 0 rz -88.32 deg; joints [3.164, 10.373, -18.087, 11.787, -16.98, -14.713]
  MoveL 1796 to (96.66, 2354.9, 513.19) mm, rotated rx 180 ry 0 rz -88.32 deg; joints [3.184, 10.502, -17.94, 11.823, -17.001, -14.76]
  MoveL 1797 to (97.51, 2357.62, 513.19) mm, rotated rx 180 ry 0 rz -88.32 deg; joints [3.205, 10.632, -17.793, 11.859, -17.022, -14.808]
  MoveL 1798 to (98.37, 2360.34, 513.19) mm, rotated rx -180 ry 0 rz -88.32 deg; joints [3.225, 10.762, -17.645, 11.895, -17.043, -14.856]
  MoveL 1799 to (99.24, 2363.05, 513.19) mm, rotated rx 180 ry 0 rz -88.32 deg; joints [3.246, 10.891, -17.498, 11.931, -17.065, -14.904]
  MoveL 1800 to (100.12, 2365.76, 513.19) mm, rotated rx -180 ry 0 rz -88.32 deg; joints [3.267, 11.021, -17.35, 11.967, -17.087, -14.952]
  MoveL 1801 to (101.01, 2368.47, 513.19) mm, rotated rx 180 ry 0 rz -88.32 deg; joints [3.288, 11.15, -17.202, 12.003, -17.108, -15.001]
  MoveL 1802 to (101.9, 2371.18, 513.19) mm, rotated rx -180 ry 0 rz -88.32 deg; joints [3.309, 11.279, -17.054, 12.04, -17.131, -15.05]
  MoveL 1803 to (102.8, 2373.88, 513.19) mm, rotated rx -180 ry 0 rz -88.32 deg; joints [3.33, 11.408, -16.907, 12.077, -17.153, -15.099]
  MoveL 1804 to (103.71, 2376.58, 513.19) mm, rotated rx 180 ry 0 rz -88.32 deg; joints [3.352, 11.537, -16.759, 12.114, -17.176, -15.148]
  MoveL 1805 to (104.62, 2379.28, 513.19) mm, rotated rx 180 ry 0 rz -88.32 deg; joints [3.374, 11.666, -16.611, 12.151, -17.198, -15.198]
  MoveL 1806 to (105.55, 2381.98, 513.19) mm, rotated rx 180 ry 0 rz -88.32 deg; joints [3.395, 11.794, -16.463, 12.188, -17.221, -15.248]
  MoveL 1807 to (106.48, 2384.67, 513.19) mm, rotated rx 180 ry 0 rz -88.32 deg; joints [3.418, 11.923, -16.315, 12.225, -17.245, -15.298]
  MoveL 1808 to (107.42, 2387.36, 513.19) mm, rotated rx -180 ry 0 rz -88.32 deg; joints [3.44, 12.051, -16.166, 12.263, -17.268, -15.348]
  MoveL 1809 to (108.36, 2390.05, 513.19) mm, rotated rx -180 ry 0 rz -88.32 deg; joints [3.462, 12.179, -16.018, 12.301, -17.292, -15.398]
  MoveL 1810 to (109.32, 2392.73, 513.19) mm, rotated rx -180 ry 0 rz -88.32 deg; joints [3.485, 12.308, -15.87, 12.338, -17.316, -15.449]
  MoveL 1811 to (110.28, 2395.42, 513.19) mm, rotated rx 180 ry 0 rz -88.32 deg; joints [3.507, 12.436, -15.721, 12.376, -17.34, -15.5]
  MoveL 1812 to (111.25, 2398.1, 513.19) mm, rotated rx -180 ry 0 rz -88.32 deg; joints [3.53, 12.563, -15.573, 12.414, -17.364, -15.551]
  MoveL 1813 to (112.22, 2400.78, 513.19) mm, rotated rx 180 ry 0 rz -88.32 deg; joints [3.553, 12.691, -15.424, 12.452, -17.389, -15.602]
  MoveL 1814 to (113.21, 2403.45, 513.19) mm, rotated rx -180 ry 0 rz -88.32 deg; joints [3.576, 12.819, -15.276, 12.491, -17.414, -15.654]
  MoveL 1815 to (114.2, 2406.12, 513.19) mm, rotated rx 180 ry 0 rz -88.32 deg; joints [3.599, 12.946, -15.127, 12.529, -17.439, -15.706]
  MoveL 1816 to (115.2, 2408.79, 513.19) mm, rotated rx -180 ry 0 rz -88.32 deg; joints [3.623, 13.074, -14.979, 12.568, -17.464, -15.758]
  MoveL 1817 to (116.2, 2411.46, 513.19) mm, rotated rx -180 ry 0 rz -88.32 deg; joints [3.646, 13.201, -14.83, 12.606, -17.49, -15.81]
  MoveL 1818 to (117.22, 2414.12, 513.19) mm, rotated rx 180 ry 0 rz -88.32 deg; joints [3.67, 13.328, -14.681, 12.645, -17.515, -15.862]
  MoveL 1819 to (118.24, 2416.78, 513.19) mm, rotated rx -180 ry 0 rz -88.32 deg; joints [3.694, 13.456, -14.532, 12.684, -17.541, -15.914]
  MoveL 1820 to (119.27, 2419.44, 513.19) mm, rotated rx 180 ry 0 rz -88.32 deg; joints [3.718, 13.582, -14.383, 12.723, -17.567, -15.967]
  MoveL 1821 to (120.3, 2422.09, 513.19) mm, rotated rx -180 ry 0 rz -88.32 deg; joints [3.742, 13.709, -14.234, 12.762, -17.594, -16.02]
  MoveL 1822 to (121.35, 2424.75, 513.19) mm, rotated rx -180 ry 0 rz -88.32 deg; joints [3.767, 13.836, -14.085, 12.801, -17.62, -16.073]
  MoveL 1823 to (122.4, 2427.4, 513.19) mm, rotated rx -180 ry 0 rz -88.32 deg; joints [3.791, 13.963, -13.936, 12.84, -17.647, -16.126]
  MoveL 1824 to (123.46, 2430.04, 513.19) mm, rotated rx 180 ry 0 rz -88.32 deg; joints [3.816, 14.089, -13.786, 12.879, -17.674, -16.179]
  MoveL 1825 to (124.52, 2432.68, 513.19) mm, rotated rx 180 ry 0 rz -88.32 deg; joints [3.841, 14.216, -13.637, 12.919, -17.701, -16.233]
  MoveL 1826 to (125.59, 2435.32, 513.19) mm, rotated rx 180 ry 0 rz -88.32 deg; joints [3.866, 14.342, -13.488, 12.958, -17.729, -16.287]
  MoveL 1827 to (126.67, 2437.96, 513.19) mm, rotated rx 180 ry 0 rz -88.32 deg; joints [3.891, 14.468, -13.338, 12.998, -17.756, -16.34]
  MoveL 1828 to (127.76, 2440.6, 513.19) mm, rotated rx -180 ry 0 rz -88.32 deg; joints [3.916, 14.594, -13.189, 13.037, -17.784, -16.394]
  MoveL 1829 to (128.86, 2443.23, 513.19) mm, rotated rx 180 ry 0 rz -88.32 deg; joints [3.941, 14.72, -13.039, 13.077, -17.812, -16.448]
  MoveL 1830 to (129.96, 2445.85, 513.19) mm, rotated rx -180 ry 0 rz -88.32 deg; joints [3.967, 14.846, -12.89, 13.117, -17.84, -16.503]
  MoveL 1831 to (131.07, 2448.48, 513.19) mm, rotated rx 180 ry 0 rz -88.32 deg; joints [3.992, 14.972, -12.74, 13.157, -17.869, -16.557]
  MoveL 1832 to (132.19, 2451.1, 513.19) mm, rotated rx 180 ry 0 rz -88.32 deg; joints [4.018, 15.097, -12.59, 13.196, -17.898, -16.612]
  MoveL 1833 to (133.31, 2453.72, 513.19) mm, rotated rx 180 ry 0 rz -88.32 deg; joints [4.044, 15.223, -12.441, 13.236, -17.926, -16.666]
  MoveL 1834 to (134.44, 2456.33, 513.19) mm, rotated rx -180 ry 0 rz -88.32 deg; joints [4.07, 15.348, -12.291, 13.276, -17.956, -16.721]
  MoveL 1835 to (135.58, 2458.95, 513.19) mm, rotated rx 180 ry 0 rz -88.32 deg; joints [4.096, 15.474, -12.141, 13.317, -17.985, -16.776]
  MoveL 1836 to (136.73, 2461.56, 513.19) mm, rotated rx 180 ry 0 rz -88.32 deg; joints [4.123, 15.599, -11.991, 13.357, -18.014, -16.831]
  MoveL 1837 to (137.89, 2464.16, 513.19) mm, rotated rx 180 ry 0 rz -88.32 deg; joints [4.149, 15.724, -11.841, 13.397, -18.044, -16.886]
  MoveL 1838 to (139.05, 2466.76, 513.19) mm, rotated rx -180 ry 0 rz -88.32 deg; joints [4.176, 15.849, -11.691, 13.437, -18.074, -16.942]
  MoveL 1839 to (140.22, 2469.36, 513.19) mm, rotated rx 180 ry 0 rz -88.32 deg; joints [4.203, 15.974, -11.541, 13.477, -18.104, -16.997]
  MoveL 1840 to (141.39, 2471.96, 513.19) mm, rotated rx 180 ry 0 rz -88.32 deg; joints [4.23, 16.098, -11.39, 13.518, -18.135, -17.053]
  MoveL 1841 to (142.57, 2474.55, 513.19) mm, rotated rx -180 ry 0 rz -88.32 deg; joints [4.257, 16.223, -11.24, 13.558, -18.165, -17.108]
  MoveL 1842 to (143.76, 2477.14, 513.19) mm, rotated rx 180 ry 0 rz -88.32 deg; joints [4.284, 16.348, -11.09, 13.599, -18.196, -17.164]
  MoveL 1843 to (144.96, 2479.73, 513.19) mm, rotated rx 180 ry 0 rz -88.32 deg; joints [4.311, 16.472, -10.939, 13.639, -18.227, -17.22]
  MoveL 1844 to (146.17, 2482.31, 513.19) mm, rotated rx 180 ry 0 rz -88.32 deg; joints [4.339, 16.596, -10.789, 13.68, -18.258, -17.276]
  MoveL 1845 to (147.38, 2484.89, 513.19) mm, rotated rx -180 ry 0 rz -88.32 deg; joints [4.366, 16.721, -10.638, 13.72, -18.289, -17.332]
  MoveL 1846 to (148.6, 2487.46, 513.19) mm, rotated rx 180 ry 0 rz -88.32 deg; joints [4.394, 16.845, -10.488, 13.761, -18.321, -17.388]
  MoveL 1847 to (149.83, 2490.04, 513.19) mm, rotated rx -180 ry 0 rz -88.32 deg; joints [4.422, 16.969, -10.337, 13.801, -18.353, -17.444]
  MoveL 1848 to (151.06, 2492.61, 513.19) mm, rotated rx -180 ry 0 rz -88.32 deg; joints [4.45, 17.093, -10.186, 13.842, -18.384, -17.501]
  MoveL 1849 to (152.3, 2495.17, 513.19) mm, rotated rx -180 ry 0 rz -88.32 deg; joints [4.478, 17.216, -10.036, 13.883, -18.417, -17.557]
  MoveL 1850 to (153.55, 2497.73, 513.19) mm, rotated rx -180 ry 0 rz -88.32 deg; joints [4.506, 17.34, -9.885, 13.923, -18.449, -17.614]
  MoveL 1851 to (154.81, 2500.29, 513.19) mm, rotated rx 180 ry 0 rz -88.32 deg; joints [4.535, 17.464, -9.734, 13.964, -18.482, -17.67]
  MoveL 1852 to (156.07, 2502.85, 513.19) mm, rotated rx -180 ry 0 rz -88.32 deg; joints [4.563, 17.587, -9.583, 14.005, -18.514, -17.727]
  MoveL 1853 to (157.34, 2505.4, 513.19) mm, rotated rx -180 ry 0 rz -88.32 deg; joints [4.592, 17.711, -9.432, 14.046, -18.547, -17.784]
  MoveL 1854 to (158.61, 2507.95, 513.19) mm, rotated rx -180 ry 0 rz -88.32 deg; joints [4.621, 17.834, -9.281, 14.086, -18.58, -17.84]
  MoveL 1855 to (159.9, 2510.49, 513.19) mm, rotated rx 180 ry 0 rz -88.32 deg; joints [4.649, 17.957, -9.13, 14.127, -18.614, -17.897]
  MoveL 1856 to (161.19, 2513.03, 513.19) mm, rotated rx -180 ry 0 rz -88.32 deg; joints [4.678, 18.08, -8.979, 14.168, -18.647, -17.954]
  MoveL 1857 to (162.49, 2515.57, 513.19) mm, rotated rx -180 ry 0 rz -88.32 deg; joints [4.708, 18.203, -8.828, 14.209, -18.681, -18.011]
  MoveL 1858 to (163.79, 2518.1, 513.19) mm, rotated rx -180 ry 0 rz -88.32 deg; joints [4.737, 18.326, -8.676, 14.249, -18.715, -18.068]
  MoveL 1859 to (165.11, 2520.63, 513.19) mm, rotated rx 180 ry 0 rz -88.32 deg; joints [4.766, 18.449, -8.525, 14.29, -18.749, -18.126]
  MoveL 1860 to (166.43, 2523.16, 513.19) mm, rotated rx -180 ry 0 rz -88.32 deg; joints [4.796, 18.571, -8.374, 14.331, -18.783, -18.183]
  MoveL 1861 to (167.75, 2525.68, 513.19) mm, rotated rx -180 ry 0 rz -88.32 deg; joints [4.825, 18.694, -8.222, 14.372, -18.818, -18.24]
  MoveL 1862 to (169.09, 2528.2, 513.19) mm, rotated rx 180 ry 0 rz -88.32 deg; joints [4.855, 18.816, -8.071, 14.413, -18.852, -18.297]
  MoveL 1863 to (170.43, 2530.71, 513.19) mm, rotated rx -180 ry 0 rz -88.32 deg; joints [4.885, 18.939, -7.919, 14.453, -18.887, -18.355]
  MoveL 1864 to (171.78, 2533.22, 513.19) mm, rotated rx -180 ry 0 rz -88.32 deg; joints [4.915, 19.061, -7.768, 14.494, -18.922, -18.412]
  MoveL 1865 to (173.13, 2535.73, 513.19) mm, rotated rx 180 ry 0 rz -88.32 deg; joints [4.945, 19.183, -7.616, 14.535, -18.958, -18.47]
  MoveL 1866 to (174.49, 2538.23, 513.19) mm, rotated rx -180 ry 0 rz -88.32 deg; joints [4.976, 19.305, -7.464, 14.576, -18.993, -18.527]
  MoveL 1867 to (175.86, 2540.73, 513.19) mm, rotated rx -180 ry 0 rz -88.32 deg; joints [5.006, 19.427, -7.313, 14.617, -19.029, -18.585]
  MoveL 1868 to (177.24, 2543.23, 513.19) mm, rotated rx 180 ry 0 rz -88.32 deg; joints [5.036, 19.549, -7.161, 14.657, -19.065, -18.643]
  MoveL 1869 to (178.62, 2545.72, 513.19) mm, rotated rx -180 ry 0 rz -88.32 deg; joints [5.067, 19.671, -7.009, 14.698, -19.101, -18.7]
  MoveL 1870 to (180.01, 2548.21, 513.19) mm, rotated rx 180 ry 0 rz -88.32 deg; joints [5.098, 19.793, -6.857, 14.739, -19.137, -18.758]
  MoveL 1871 to (181.41, 2550.69, 513.19) mm, rotated rx -180 ry 0 rz -88.32 deg; joints [5.129, 19.914, -6.705, 14.78, -19.173, -18.816]
  MoveL 1872 to (182.81, 2553.17, 513.19) mm, rotated rx 180 ry 0 rz -88.32 deg; joints [5.16, 20.036, -6.553, 14.82, -19.21, -18.873]
  MoveL 1873 to (184.22, 2555.65, 513.19) mm, rotated rx -180 ry 0 rz -88.32 deg; joints [5.191, 20.157, -6.401, 14.861, -19.246, -18.931]
  MoveL 1874 to (185.64, 2558.12, 513.19) mm, rotated rx -180 ry 0 rz -88.32 deg; joints [5.222, 20.279, -6.249, 14.901, -19.283, -18.989]
  MoveL 1875 to (187.06, 2560.59, 513.19) mm, rotated rx -180 ry 0 rz -88.32 deg; joints [5.253, 20.4, -6.097, 14.942, -19.32, -19.047]
  MoveL 1876 to (188.5, 2563.05, 513.19) mm, rotated rx -180 ry 0 rz -88.32 deg; joints [5.285, 20.521, -5.945, 14.983, -19.358, -19.105]
  MoveL 1877 to (189.93, 2565.51, 513.19) mm, rotated rx -180 ry 0 rz -88.32 deg; joints [5.316, 20.642, -5.792, 15.023, -19.395, -19.163]
  MoveL 1878 to (191.38, 2567.97, 513.19) mm, rotated rx -180 ry 0 rz -88.32 deg; joints [5.348, 20.763, -5.64, 15.064, -19.433, -19.221]
  MoveL 1879 to (192.83, 2570.42, 513.19) mm, rotated rx 180 ry 0 rz -88.32 deg; joints [5.38, 20.884, -5.488, 15.104, -19.471, -19.279]
  MoveL 1880 to (194.29, 2572.87, 513.19) mm, rotated rx -180 ry 0 rz -88.32 deg; joints [5.412, 21.004, -5.335, 15.145, -19.509, -19.337]
  MoveL 1881 to (195.76, 2575.31, 513.19) mm, rotated rx -180 ry 0 rz -88.32 deg; joints [5.444, 21.125, -5.183, 15.185, -19.547, -19.395]
  MoveL 1882 to (197.23, 2577.75, 513.19) mm, rotated rx -180 ry 0 rz -88.32 deg; joints [5.476, 21.246, -5.03, 15.226, -19.586, -19.452]
  MoveL 1883 to (198.71, 2580.19, 513.19) mm, rotated rx 180 ry 0 rz -88.32 deg; joints [5.508, 21.366, -4.878, 15.266, -19.624, -19.51]
  MoveL 1884 to (200.2, 2582.62, 513.19) mm, rotated rx -180 ry 0 rz -88.32 deg; joints [5.541, 21.487, -4.725, 15.306, -19.663, -19.568]
  MoveL 1885 to (201.69, 2585.05, 513.19) mm, rotated rx 180 ry 0 rz -88.32 deg; joints [5.573, 21.607, -4.572, 15.347, -19.702, -19.626]
  MoveL 1886 to (203.19, 2587.47, 513.19) mm, rotated rx -180 ry 0 rz -88.32 deg; joints [5.606, 21.727, -4.42, 15.387, -19.741, -19.685]
  MoveL 1887 to (204.7, 2589.89, 513.19) mm, rotated rx -180 ry 0 rz -88.32 deg; joints [5.638, 21.847, -4.267, 15.427, -19.78, -19.743]
  MoveL 1888 to (206.21, 2592.3, 513.19) mm, rotated rx -180 ry 0 rz -88.32 deg; joints [5.671, 21.967, -4.114, 15.467, -19.82, -19.801]
  MoveL 1889 to (207.73, 2594.71, 513.19) mm, rotated rx -180 ry 0 rz -88.32 deg; joints [5.704, 22.087, -3.961, 15.507, -19.859, -19.859]
  MoveL 1890 to (209.26, 2597.12, 513.19) mm, rotated rx -180 ry 0 rz -88.32 deg; joints [5.737, 22.207, -3.808, 15.547, -19.899, -19.917]
  MoveL 1891 to (210.79, 2599.52, 513.19) mm, rotated rx 180 ry 0 rz -88.32 deg; joints [5.77, 22.327, -3.655, 15.587, -19.939, -19.975]
  MoveL 1892 to (212.33, 2601.92, 513.19) mm, rotated rx -180 ry 0 rz -88.32 deg; joints [5.803, 22.446, -3.502, 15.627, -19.979, -20.033]
  MoveL 1893 to (213.88, 2604.31, 513.19) mm, rotated rx -180 ry 0 rz -88.32 deg; joints [5.837, 22.566, -3.349, 15.667, -20.02, -20.091]
  MoveL 1894 to (215.44, 2606.7, 513.19) mm, rotated rx -180 ry 0 rz -88.32 deg; joints [5.87, 22.686, -3.196, 15.707, -20.06, -20.149]
  MoveL 1895 to (217, 2609.08, 513.19) mm, rotated rx -180 ry 0 rz -88.32 deg; joints [5.904, 22.805, -3.043, 15.747, -20.101, -20.207]
  MoveL 1896 to (218.56, 2611.46, 513.19) mm, rotated rx 180 ry 0 rz -88.32 deg; joints [5.937, 22.924, -2.889, 15.787, -20.142, -20.265]
  MoveL 1897 to (220.14, 2613.84, 513.19) mm, rotated rx -180 ry 0 rz -88.32 deg; joints [5.971, 23.043, -2.736, 15.826, -20.183, -20.322]
  MoveL 1898 to (221.72, 2616.21, 513.19) mm, rotated rx -180 ry 0 rz -88.32 deg; joints [6.005, 23.163, -2.583, 15.866, -20.224, -20.38]
  MoveL 1899 to (223.31, 2618.58, 513.19) mm, rotated rx -180 ry 0 rz -88.32 deg; joints [6.039, 23.282, -2.429, 15.906, -20.266, -20.438]
  MoveL 1900 to (224.9, 2620.94, 513.19) mm, rotated rx -180 ry 0 rz -88.32 deg; joints [6.073, 23.401, -2.276, 15.945, -20.307, -20.496]
  MoveL 1901 to (226.5, 2623.3, 513.19) mm, rotated rx -180 ry 0 rz -88.32 deg; joints [6.107, 23.52, -2.122, 15.985, -20.349, -20.554]
  MoveL 1902 to (228.11, 2625.65, 513.19) mm, rotated rx -180 ry 0 rz -88.32 deg; joints [6.142, 23.638, -1.969, 16.024, -20.391, -20.612]
  MoveL 1903 to (229.72, 2628, 513.19) mm, rotated rx -180 ry 0 rz -88.32 deg; joints [6.176, 23.757, -1.815, 16.063, -20.433, -20.67]
  MoveL 1904 to (231.34, 2630.34, 513.19) mm, rotated rx 180 ry 0 rz -88.32 deg; joints [6.21, 23.876, -1.662, 16.103, -20.475, -20.728]
  MoveL 1905 to (232.97, 2632.68, 513.19) mm, rotated rx -180 ry 0 rz -88.32 deg; joints [6.245, 23.994, -1.508, 16.142, -20.517, -20.785]
  MoveL 1906 to (234.61, 2635.02, 513.19) mm, rotated rx 180 ry 0 rz -88.32 deg; joints [6.28, 24.113, -1.354, 16.181, -20.56, -20.843]
  MoveL 1907 to (236.25, 2637.35, 513.19) mm, rotated rx 180 ry 0 rz -88.32 deg; joints [6.315, 24.231, -1.2, 16.22, -20.603, -20.901]
  MoveL 1908 to (237.89, 2639.68, 513.19) mm, rotated rx 180 ry 0 rz -88.32 deg; joints [6.349, 24.349, -1.047, 16.259, -20.646, -20.959]
  MoveL 1909 to (239.55, 2642, 513.19) mm, rotated rx -180 ry 0 rz -88.32 deg; joints [6.384, 24.468, -0.893, 16.298, -20.689, -21.016]
  MoveL 1910 to (241.21, 2644.31, 513.19) mm, rotated rx 180 ry 0 rz -88.32 deg; joints [6.42, 24.586, -0.739, 16.337, -20.732, -21.074]
  MoveL 1911 to (242.87, 2646.63, 513.19) mm, rotated rx 180 ry 0 rz -88.32 deg; joints [6.455, 24.704, -0.585, 16.376, -20.776, -21.132]
  MoveL 1912 to (244.54, 2648.93, 513.19) mm, rotated rx -180 ry 0 rz -88.32 deg; joints [6.49, 24.822, -0.431, 16.415, -20.819, -21.189]
  MoveL 1913 to (246.22, 2651.23, 513.19) mm, rotated rx 180 ry 0 rz -88.32 deg; joints [6.525, 24.94, -0.277, 16.453, -20.863, -21.247]
  MoveL 1914 to (247.91, 2653.53, 513.19) mm, rotated rx -180 ry 0 rz -88.32 deg; joints [6.561, 25.058, -0.123, 16.492, -20.907, -21.304]
  MoveL 1915 to (249.6, 2655.83, 513.19) mm, rotated rx 180 ry 0 rz -88.32 deg; joints [6.596, 25.175, 0.032, 16.531, -20.951, -21.362]
  MoveL 1916 to (251.3, 2658.11, 513.19) mm, rotated rx -180 ry 0 rz -88.32 deg; joints [6.632, 25.293, 0.186, 16.569, -20.995, -21.419]
  MoveL 1917 to (253, 2660.4, 513.19) mm, rotated rx 180 ry 0 rz -88.32 deg; joints [6.668, 25.41, 0.34, 16.607, -21.04, -21.476]
  MoveL 1918 to (254.72, 2662.68, 513.19) mm, rotated rx -180 ry 0 rz -88.32 deg; joints [6.704, 25.528, 0.494, 16.646, -21.084, -21.534]
  MoveL 1919 to (256.43, 2664.95, 513.19) mm, rotated rx -180 ry 0 rz -88.32 deg; joints [6.74, 25.645, 0.649, 16.684, -21.129, -21.591]
  MoveL 1920 to (258.16, 2667.22, 513.19) mm, rotated rx 180 ry 0 rz -88.32 deg; joints [6.776, 25.763, 0.803, 16.722, -21.174, -21.648]
  MoveL 1921 to (259.89, 2669.48, 513.19) mm, rotated rx 180 ry 0 rz -88.32 deg; joints [6.812, 25.88, 0.958, 16.76, -21.219, -21.706]
  MoveL 1922 to (261.63, 2671.74, 513.19) mm, rotated rx -180 ry 0 rz -88.32 deg; joints [6.848, 25.997, 1.112, 16.798, -21.264, -21.763]
  MoveL 1923 to (263.37, 2674, 513.19) mm, rotated rx -180 ry 0 rz -88.32 deg; joints [6.885, 26.114, 1.267, 16.836, -21.309, -21.82]
  MoveL 1924 to (265.12, 2676.25, 513.19) mm, rotated rx -180 ry 0 rz -88.32 deg; joints [6.921, 26.231, 1.421, 16.874, -21.355, -21.877]
  MoveL 1925 to (266.87, 2678.49, 513.19) mm, rotated rx 180 ry 0 rz -88.32 deg; joints [6.958, 26.348, 1.576, 16.912, -21.401, -21.934]
  MoveL 1926 to (268.64, 2680.73, 513.19) mm, rotated rx 180 ry 0 rz -88.32 deg; joints [6.994, 26.465, 1.73, 16.95, -21.446, -21.991]
  MoveL 1927 to (270.4, 2682.97, 513.19) mm, rotated rx 180 ry 0 rz -88.32 deg; joints [7.031, 26.582, 1.885, 16.987, -21.492, -22.048]
  MoveL 1928 to (272.18, 2685.2, 513.19) mm, rotated rx -180 ry 0 rz -88.32 deg; joints [7.068, 26.699, 2.04, 17.025, -21.539, -22.105]
  MoveL 1929 to (273.96, 2687.42, 513.19) mm, rotated rx 180 ry 0 rz -88.32 deg; joints [7.105, 26.815, 2.195, 17.062, -21.585, -22.161]
  MoveL 1930 to (275.75, 2689.64, 513.19) mm, rotated rx 180 ry 0 rz -88.32 deg; joints [7.142, 26.932, 2.35, 17.099, -21.631, -22.218]
  MoveL 1931 to (277.54, 2691.86, 513.19) mm, rotated rx 180 ry 0 rz -88.32 deg; joints [7.179, 27.048, 2.504, 17.137, -21.678, -22.275]
  MoveL 1932 to (279.34, 2694.07, 513.19) mm, rotated rx 180 ry 0 rz -88.32 deg; joints [7.216, 27.165, 2.659, 17.174, -21.725, -22.332]
  MoveL 1933 to (281.15, 2696.27, 513.19) mm, rotated rx 180 ry 0 rz -88.32 deg; joints [7.253, 27.281, 2.814, 17.211, -21.772, -22.388]
  MoveL 1934 to (282.96, 2698.47, 513.19) mm, rotated rx -180 ry 0 rz -88.32 deg; joints [7.29, 27.397, 2.969, 17.248, -21.819, -22.445]
  MoveL 1935 to (284.78, 2700.67, 513.19) mm, rotated rx -180 ry 0 rz -88.32 deg; joints [7.328, 27.513, 3.125, 17.285, -21.866, -22.501]
  MoveL 1936 to (286.6, 2702.86, 513.19) mm, rotated rx 180 ry 0 rz -88.32 deg; joints [7.365, 27.63, 3.28, 17.322, -21.914, -22.558]
  MoveL 1937 to (288.43, 2705.04, 513.19) mm, rotated rx -180 ry 0 rz -88.32 deg; joints [7.403, 27.746, 3.435, 17.359, -21.961, -22.614]
  MoveL 1938 to (290.27, 2707.22, 513.19) mm, rotated rx 180 ry 0 rz -88.32 deg; joints [7.441, 27.862, 3.59, 17.395, -22.009, -22.67]
  MoveL 1939 to (292.11, 2709.39, 513.19) mm, rotated rx -180 ry 0 rz -88.32 deg; joints [7.479, 27.977, 3.745, 17.432, -22.057, -22.726]
  MoveL 1940 to (293.96, 2711.56, 513.19) mm, rotated rx -180 ry 0 rz -88.32 deg; joints [7.516, 28.093, 3.901, 17.469, -22.105, -22.783]
  MoveL 1941 to (295.81, 2713.73, 513.19) mm, rotated rx -180 ry 0 rz -88.32 deg; joints [7.554, 28.209, 4.056, 17.505, -22.153, -22.839]
  MoveL 1942 to (297.67, 2715.88, 513.19) mm, rotated rx -180 ry 0 rz -88.32 deg; joints [7.592, 28.325, 4.211, 17.541, -22.201, -22.895]
  MoveL 1943 to (299.54, 2718.04, 513.19) mm, rotated rx -180 ry 0 rz -88.32 deg; joints [7.631, 28.44, 4.367, 17.578, -22.25, -22.951]
  MoveL 1944 to (301.41, 2720.19, 513.19) mm, rotated rx -180 ry 0 rz -88.32 deg; joints [7.669, 28.556, 4.522, 17.614, -22.298, -23.007]
  MoveL 1945 to (303.29, 2722.33, 513.19) mm, rotated rx 180 ry 0 rz -88.32 deg; joints [7.707, 28.671, 4.678, 17.65, -22.347, -23.062]
  MoveL 1946 to (305.18, 2724.47, 513.19) mm, rotated rx -180 ry 0 rz -88.32 deg; joints [7.745, 28.787, 4.833, 17.686, -22.396, -23.118]
  MoveL 1947 to (307.07, 2726.6, 513.19) mm, rotated rx 180 ry 0 rz -88.32 deg; joints [7.784, 28.902, 4.989, 17.722, -22.445, -23.174]
  MoveL 1948 to (308.96, 2728.73, 513.19) mm, rotated rx 180 ry 0 rz -88.32 deg; joints [7.823, 29.017, 5.145, 17.757, -22.495, -23.23]
  MoveL 1949 to (310.87, 2730.85, 513.19) mm, rotated rx -180 ry 0 rz -88.32 deg; joints [7.861, 29.133, 5.3, 17.793, -22.544, -23.285]
  MoveL 1950 to (312.78, 2732.96, 513.19) mm, rotated rx 180 ry 0 rz -88.32 deg; joints [7.9, 29.248, 5.456, 17.829, -22.593, -23.341]
  MoveL 1951 to (314.69, 2735.07, 513.19) mm, rotated rx -180 ry 0 rz -88.32 deg; joints [7.939, 29.363, 5.612, 17.864, -22.643, -23.396]
  MoveL 1952 to (316.61, 2737.18, 513.19) mm, rotated rx -180 ry 0 rz -88.32 deg; joints [7.978, 29.478, 5.768, 17.9, -22.693, -23.451]
  MoveL 1953 to (318.54, 2739.28, 513.19) mm, rotated rx -180 ry 0 rz -88.32 deg; joints [8.017, 29.593, 5.924, 17.935, -22.743, -23.507]
  MoveL 1954 to (320.47, 2741.37, 513.19) mm, rotated rx 180 ry 0 rz -88.32 deg; joints [8.056, 29.707, 6.08, 17.97, -22.793, -23.562]
  MoveL 1955 to (322.41, 2743.46, 513.19) mm, rotated rx 180 ry 0 rz -88.32 deg; joints [8.095, 29.822, 6.236, 18.005, -22.843, -23.617]
  MoveL 1956 to (324.35, 2745.55, 513.19) mm, rotated rx 180 ry 0 rz -88.32 deg; joints [8.134, 29.937, 6.392, 18.04, -22.894, -23.672]
  MoveL 1957 to (326.3, 2747.63, 513.19) mm, rotated rx -180 ry 0 rz -88.32 deg; joints [8.173, 30.052, 6.548, 18.075, -22.944, -23.727]
  MoveL 1958 to (328.26, 2749.7, 513.19) mm, rotated rx 180 ry 0 rz -88.32 deg; joints [8.213, 30.166, 6.704, 18.11, -22.995, -23.782]
  MoveL 1959 to (330.22, 2751.77, 513.19) mm, rotated rx -180 ry 0 rz -88.32 deg; joints [8.252, 30.281, 6.86, 18.145, -23.046, -23.837]
  MoveL 1960 to (332.19, 2753.83, 513.19) mm, rotated rx 180 ry 0 rz -88.32 deg; joints [8.292, 30.395, 7.016, 18.18, -23.097, -23.892]
  MoveL 1961 to (334.16, 2755.88, 513.19) mm, rotated rx -180 ry 0 rz -88.32 deg; joints [8.331, 30.509, 7.173, 18.214, -23.148, -23.946]
  MoveL 1962 to (336.14, 2757.93, 513.19) mm, rotated rx -180 ry 0 rz -88.32 deg; joints [8.371, 30.624, 7.329, 18.249, -23.199, -24.001]
  MoveL 1963 to (338.12, 2759.98, 513.19) mm, rotated rx -180 ry 0 rz -88.32 deg; joints [8.411, 30.738, 7.485, 18.283, -23.251, -24.055]
  MoveL 1964 to (340.11, 2762.02, 513.19) mm, rotated rx 180 ry 0 rz -88.32 deg; joints [8.451, 30.852, 7.642, 18.317, -23.302, -24.11]
  MoveL 1965 to (342.11, 2764.05, 513.19) mm, rotated rx -180 ry 0 rz -88.32 deg; joints [8.49, 30.966, 7.798, 18.352, -23.354, -24.164]
  MoveL 1966 to (344.11, 2766.08, 513.19) mm, rotated rx 180 ry 0 rz -88.32 deg; joints [8.53, 31.08, 7.954, 18.386, -23.406, -24.219]
  MoveL 1967 to (346.12, 2768.1, 513.19) mm, rotated rx 180 ry 0 rz -88.32 deg; joints [8.571, 31.194, 8.111, 18.42, -23.458, -24.273]
  MoveL 1968 to (348.13, 2770.12, 513.19) mm, rotated rx 180 ry 0 rz -88.32 deg; joints [8.611, 31.308, 8.267, 18.454, -23.51, -24.327]
  MoveL 1969 to (350.15, 2772.13, 513.19) mm, rotated rx 180 ry 0 rz -88.32 deg; joints [8.651, 31.422, 8.424, 18.488, -23.562, -24.381]
  MoveL 1970 to (352.18, 2774.14, 513.19) mm, rotated rx -180 ry 0 rz -88.32 deg; joints [8.691, 31.536, 8.581, 18.521, -23.615, -24.435]
  MoveL 1971 to (354.21, 2776.14, 513.19) mm, rotated rx -180 ry 0 rz -88.32 deg; joints [8.732, 31.65, 8.737, 18.555, -23.667, -24.489]
  MoveL 1972 to (356.24, 2778.13, 513.19) mm, rotated rx -180 ry 0 rz -88.32 deg; joints [8.772, 31.763, 8.894, 18.588, -23.72, -24.543]
  MoveL 1973 to (358.28, 2780.12, 513.19) mm, rotated rx -180 ry 0 rz -88.32 deg; joints [8.813, 31.877, 9.051, 18.622, -23.773, -24.596]
  MoveL 1974 to (360.33, 2782.11, 513.19) mm, rotated rx 180 ry 0 rz -88.32 deg; joints [8.853, 31.99, 9.208, 18.655, -23.826, -24.65]
  MoveL 1975 to (362.38, 2784.08, 513.19) mm, rotated rx 180 ry 0 rz -88.32 deg; joints [8.894, 32.104, 9.365, 18.688, -23.879, -24.704]
  MoveL 1976 to (364.44, 2786.05, 513.19) mm, rotated rx -180 ry 0 rz -88.32 deg; joints [8.935, 32.217, 9.521, 18.722, -23.932, -24.757]
  MoveL 1977 to (366.5, 2788.02, 513.19) mm, rotated rx -180 ry 0 rz -88.32 deg; joints [8.976, 32.331, 9.678, 18.755, -23.985, -24.81]
  MoveL 1978 to (368.57, 2789.98, 513.19) mm, rotated rx -180 ry 0 rz -88.32 deg; joints [9.016, 32.444, 9.835, 18.788, -24.039, -24.864]
  MoveL 1979 to (370.65, 2791.93, 513.19) mm, rotated rx -180 ry 0 rz -88.32 deg; joints [9.057, 32.557, 9.992, 18.82, -24.092, -24.917]
  MoveL 1980 to (372.73, 2793.88, 513.19) mm, rotated rx -180 ry 0 rz -88.32 deg; joints [9.098, 32.67, 10.15, 18.853, -24.146, -24.97]
  MoveL 1981 to (374.81, 2795.83, 513.19) mm, rotated rx -180 ry 0 rz -88.32 deg; joints [9.14, 32.784, 10.307, 18.886, -24.2, -25.023]
  MoveL 1982 to (376.9, 2797.76, 513.19) mm, rotated rx -180 ry 0 rz -88.32 deg; joints [9.181, 32.897, 10.464, 18.918, -24.254, -25.076]
  MoveL 1983 to (379, 2799.69, 513.19) mm, rotated rx 180 ry 0 rz -88.32 deg; joints [9.222, 33.01, 10.621, 18.951, -24.308, -25.129]
  MoveL 1984 to (381.1, 2801.62, 513.19) mm, rotated rx 180 ry 0 rz -88.32 deg; joints [9.263, 33.123, 10.778, 18.983, -24.363, -25.182]
  MoveL 1985 to (383.21, 2803.54, 513.19) mm, rotated rx 180 ry 0 rz -88.32 deg; joints [9.305, 33.236, 10.936, 19.016, -24.417, -25.234]
  MoveL 1986 to (385.32, 2805.45, 513.19) mm, rotated rx 180 ry 0 rz -88.32 deg; joints [9.346, 33.348, 11.093, 19.048, -24.472, -25.287]
  MoveL 1987 to (387.44, 2807.36, 513.19) mm, rotated rx 180 ry 0 rz -88.32 deg; joints [9.388, 33.461, 11.25, 19.08, -24.527, -25.34]
  MoveL 1988 to (389.56, 2809.26, 513.19) mm, rotated rx 180 ry 0 rz -88.32 deg; joints [9.43, 33.574, 11.408, 19.112, -24.581, -25.392]
  MoveL 1989 to (391.69, 2811.15, 513.19) mm, rotated rx 180 ry 0 rz -88.32 deg; joints [9.471, 33.686, 11.565, 19.144, -24.636, -25.444]
  MoveL 1990 to (393.82, 2813.04, 513.19) mm, rotated rx -180 ry 0 rz -88.32 deg; joints [9.513, 33.799, 11.723, 19.175, -24.691, -25.497]
  MoveL 1991 to (395.96, 2814.92, 513.19) mm, rotated rx -180 ry 0 rz -88.32 deg; joints [9.555, 33.912, 11.88, 19.207, -24.747, -25.549]
  MoveL 1992 to (398.11, 2816.8, 513.19) mm, rotated rx 180 ry 0 rz -88.32 deg; joints [9.597, 34.024, 12.038, 19.239, -24.802, -25.601]
  MoveL 1993 to (400.25, 2818.67, 513.19) mm, rotated rx 180 ry 0 rz -88.32 deg; joints [9.639, 34.137, 12.196, 19.27, -24.858, -25.653]
  MoveL 1994 to (402.41, 2820.54, 513.19) mm, rotated rx 180 ry 0 rz -88.32 deg; joints [9.681, 34.249, 12.353, 19.302, -24.913, -25.705]
  MoveL 1995 to (404.57, 2822.4, 513.19) mm, rotated rx 180 ry 0 rz -88.32 deg; joints [9.723, 34.361, 12.511, 19.333, -24.969, -25.757]
  MoveL 1996 to (406.73, 2824.25, 513.19) mm, rotated rx 180 ry 0 rz -88.32 deg; joints [9.765, 34.474, 12.669, 19.364, -25.025, -25.808]
  MoveL 1997 to (408.9, 2826.1, 513.19) mm, rotated rx 180 ry 0 rz -88.32 deg; joints [9.807, 34.586, 12.827, 19.395, -25.081, -25.86]
  MoveL 1998 to (411.08, 2827.94, 513.19) mm, rotated rx -180 ry 0 rz -88.32 deg; joints [9.85, 34.698, 12.984, 19.426, -25.137, -25.912]
  MoveL 1999 to (413.26, 2829.77, 513.19) mm, rotated rx -180 ry 0 rz -88.32 deg; joints [9.892, 34.81, 13.142, 19.457, -25.194, -25.963]
  MoveL 2000 to (415.45, 2831.6, 513.19) mm, rotated rx 180 ry 0 rz -88.32 deg; joints [9.934, 34.922, 13.3, 19.488, -25.25, -26.015]
  MoveL 2001 to (417.64, 2833.42, 513.19) mm, rotated rx 180 ry 0 rz -88.32 deg; joints [9.977, 35.034, 13.458, 19.519, -25.307, -26.066]
  MoveL 2002 to (419.83, 2835.24, 513.19) mm, rotated rx -180 ry 0 rz -88.32 deg; joints [10.019, 35.146, 13.616, 19.549, -25.363, -26.117]
  MoveL 2003 to (422.04, 2837.05, 513.19) mm, rotated rx -180 ry 0 rz -88.32 deg; joints [10.062, 35.258, 13.774, 19.58, -25.42, -26.168]
  MoveL 2004 to (424.24, 2838.85, 513.19) mm, rotated rx -180 ry 0 rz -88.32 deg; joints [10.105, 35.37, 13.933, 19.61, -25.477, -26.219]
  MoveL 2005 to (426.45, 2840.65, 513.19) mm, rotated rx -180 ry 0 rz -88.32 deg; joints [10.148, 35.481, 14.091, 19.641, -25.534, -26.27]
  MoveL 2006 to (428.67, 2842.44, 513.19) mm, rotated rx -180 ry 0 rz -88.32 deg; joints [10.19, 35.593, 14.249, 19.671, -25.591, -26.321]
  MoveL 2007 to (430.89, 2844.23, 513.19) mm, rotated rx -180 ry 0 rz -88.32 deg; joints [10.233, 35.705, 14.407, 19.701, -25.649, -26.372]
  MoveL 2008 to (433.12, 2846.01, 513.19) mm, rotated rx 180 ry 0 rz -88.32 deg; joints [10.276, 35.816, 14.566, 19.731, -25.706, -26.422]
  MoveL 2009 to (435.35, 2847.78, 513.19) mm, rotated rx 180 ry 0 rz -88.32 deg; joints [10.319, 35.928, 14.724, 19.761, -25.764, -26.473]
  MoveL 2010 to (437.58, 2849.55, 513.19) mm, rotated rx 180 ry 0 rz -88.32 deg; joints [10.362, 36.04, 14.882, 19.791, -25.821, -26.523]
  MoveL 2011 to (439.83, 2851.31, 513.19) mm, rotated rx -180 ry 0 rz -88.32 deg; joints [10.406, 36.151, 15.041, 19.821, -25.879, -26.574]
  MoveL 2012 to (442.07, 2853.06, 513.19) mm, rotated rx -180 ry 0 rz -88.32 deg; joints [10.449, 36.262, 15.199, 19.85, -25.937, -26.624]
  MoveL 2013 to (444.32, 2854.81, 513.19) mm, rotated rx -180 ry 0 rz -88.32 deg; joints [10.492, 36.374, 15.358, 19.88, -25.995, -26.674]
  MoveL 2014 to (446.58, 2856.55, 513.19) mm, rotated rx -180 ry 0 rz -88.32 deg; joints [10.535, 36.485, 15.516, 19.909, -26.053, -26.724]
  MoveL 2015 to (448.84, 2858.29, 513.19) mm, rotated rx -180 ry 0 rz -88.32 deg; joints [10.579, 36.596, 15.675, 19.939, -26.112, -26.774]
  MoveL 2016 to (451.11, 2860.02, 513.19) mm, rotated rx -180 ry 0 rz -88.32 deg; joints [10.622, 36.708, 15.834, 19.968, -26.17, -26.824]
  MoveL 2017 to (453.38, 2861.74, 513.19) mm, rotated rx -180 ry 0 rz -88.32 deg; joints [10.666, 36.819, 15.992, 19.997, -26.229, -26.874]
  MoveL 2018 to (455.65, 2863.45, 513.19) mm, rotated rx 180 ry 0 rz -88.32 deg; joints [10.709, 36.93, 16.151, 20.026, -26.287, -26.924]
  MoveL 2019 to (457.93, 2865.16, 513.19) mm, rotated rx -180 ry 0 rz -88.32 deg; joints [10.753, 37.041, 16.31, 20.055, -26.346, -26.973]
  MoveL 2020 to (460.22, 2866.87, 513.19) mm, rotated rx 180 ry 0 rz -88.32 deg; joints [10.797, 37.152, 16.469, 20.084, -26.405, -27.023]
  MoveL 2021 to (462.51, 2868.56, 513.19) mm, rotated rx -180 ry 0 rz -88.32 deg; joints [10.841, 37.263, 16.628, 20.113, -26.464, -27.072]
  MoveL 2022 to (464.8, 2870.25, 513.19) mm, rotated rx 180 ry 0 rz -88.32 deg; joints [10.884, 37.374, 16.787, 20.142, -26.523, -27.121]
  MoveL 2023 to (467.1, 2871.94, 513.19) mm, rotated rx 180 ry 0 rz -88.32 deg; joints [10.928, 37.485, 16.946, 20.171, -26.583, -27.171]
  MoveL 2024 to (469.4, 2873.61, 513.19) mm, rotated rx 180 ry 0 rz -88.32 deg; joints [10.972, 37.596, 17.105, 20.199, -26.642, -27.22]
  MoveL 2025 to (471.71, 2875.29, 513.19) mm, rotated rx 180 ry 0 rz -88.32 deg; joints [11.016, 37.707, 17.264, 20.228, -26.702, -27.269]
  MoveL 2026 to (474.02, 2876.95, 513.19) mm, rotated rx -180 ry 0 rz -88.32 deg; joints [11.06, 37.817, 17.423, 20.256, -26.761, -27.318]
  MoveL 2027 to (476.34, 2878.61, 513.19) mm, rotated rx 180 ry 0 rz -88.32 deg; joints [11.105, 37.928, 17.582, 20.284, -26.821, -27.367]
  MoveL 2028 to (478.67, 2880.26, 513.19) mm, rotated rx -180 ry 0 rz -88.32 deg; joints [11.149, 38.039, 17.741, 20.312, -26.881, -27.416]
  MoveL 2029 to (480.99, 2881.9, 513.19) mm, rotated rx 180 ry 0 rz -88.32 deg; joints [11.193, 38.149, 17.9, 20.34, -26.941, -27.464]
  MoveL 2030 to (483.32, 2883.54, 513.19) mm, rotated rx -180 ry 0 rz -88.32 deg; joints [11.237, 38.26, 18.06, 20.368, -27.001, -27.513]
  MoveL 2031 to (485.66, 2885.17, 513.19) mm, rotated rx -180 ry 0 rz -88.32 deg; joints [11.282, 38.37, 18.219, 20.396, -27.062, -27.561]
  MoveL 2032 to (488, 2886.8, 513.19) mm, rotated rx -180 ry 0 rz -88.32 deg; joints [11.326, 38.481, 18.378, 20.424, -27.122, -27.61]
  MoveL 2033 to (490.35, 2888.42, 513.19) mm, rotated rx 180 ry 0 rz -88.32 deg; joints [11.371, 38.591, 18.538, 20.452, -27.183, -27.658]
  MoveL 2034 to (492.7, 2890.03, 513.19) mm, rotated rx 180 ry 0 rz -88.32 deg; joints [11.415, 38.702, 18.697, 20.479, -27.243, -27.706]
  MoveL 2035 to (495.05, 2891.64, 513.19) mm, rotated rx 180 ry 0 rz -88.32 deg; joints [11.46, 38.812, 18.857, 20.507, -27.304, -27.754]
  MoveL 2036 to (497.41, 2893.24, 513.19) mm, rotated rx 180 ry 0 rz -88.32 deg; joints [11.504, 38.922, 19.016, 20.534, -27.365, -27.802]
  MoveL 2037 to (499.77, 2894.83, 513.19) mm, rotated rx -180 ry 0 rz -88.32 deg; joints [11.549, 39.033, 19.176, 20.562, -27.426, -27.85]
  MoveL 2038 to (502.14, 2896.41, 513.19) mm, rotated rx 180 ry 0 rz -88.32 deg; joints [11.594, 39.143, 19.336, 20.589, -27.487, -27.898]
  MoveL 2039 to (504.51, 2897.99, 513.19) mm, rotated rx 180 ry 0 rz -88.32 deg; joints [11.639, 39.253, 19.495, 20.616, -27.548, -27.946]
  MoveL 2040 to (506.89, 2899.56, 513.19) mm, rotated rx 180 ry 0 rz -88.32 deg; joints [11.684, 39.363, 19.655, 20.643, -27.609, -27.994]
  MoveL 2041 to (509.27, 2901.13, 513.19) mm, rotated rx -180 ry 0 rz -88.32 deg; joints [11.729, 39.473, 19.815, 20.67, -27.671, -28.041]
  MoveL 2042 to (511.66, 2902.69, 513.19) mm, rotated rx -180 ry 0 rz -88.32 deg; joints [11.774, 39.583, 19.975, 20.697, -27.732, -28.089]
  MoveL 2043 to (514.05, 2904.24, 513.19) mm, rotated rx -180 ry 0 rz -88.32 deg; joints [11.819, 39.693, 20.135, 20.724, -27.794, -28.136]
  MoveL 2044 to (516.44, 2905.79, 513.19) mm, rotated rx -180 ry 0 rz -88.32 deg; joints [11.864, 39.803, 20.295, 20.751, -27.856, -28.183]
  MoveL 2045 to (518.84, 2907.33, 513.19) mm, rotated rx -180 ry 0 rz -88.32 deg; joints [11.909, 39.913, 20.455, 20.777, -27.918, -28.23]
  MoveL 2046 to (521.24, 2908.86, 513.19) mm, rotated rx -180 ry 0 rz -88.32 deg; joints [11.954, 40.023, 20.615, 20.804, -27.98, -28.277]
  MoveL 2047 to (523.65, 2910.38, 513.19) mm, rotated rx -180 ry 0 rz -88.32 deg; joints [11.999, 40.133, 20.775, 20.83, -28.042, -28.324]
  MoveL 2048 to (526.06, 2911.9, 513.19) mm, rotated rx 180 ry 0 rz -88.32 deg; joints [12.045, 40.243, 20.935, 20.857, -28.104, -28.371]
  MoveL 2049 to (528.48, 2913.41, 513.19) mm, rotated rx 180 ry 0 rz -88.32 deg; joints [12.09, 40.353, 21.095, 20.883, -28.167, -28.418]
  MoveL 2050 to (530.9, 2914.92, 513.19) mm, rotated rx -180 ry 0 rz -88.32 deg; joints [12.136, 40.462, 21.255, 20.909, -28.229, -28.465]
  MoveL 2051 to (533.32, 2916.42, 513.19) mm, rotated rx -180 ry 0 rz -88.32 deg; joints [12.181, 40.572, 21.416, 20.935, -28.292, -28.511]
  MoveL 2052 to (535.75, 2917.91, 513.19) mm, rotated rx -180 ry 0 rz -88.32 deg; joints [12.227, 40.682, 21.576, 20.961, -28.354, -28.558]
  MoveL 2053 to (538.18, 2919.39, 513.19) mm, rotated rx -180 ry 0 rz -88.32 deg; joints [12.272, 40.791, 21.737, 20.987, -28.417, -28.604]
